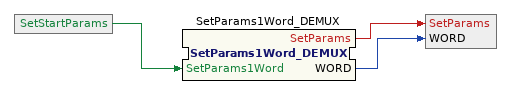
      [picture p97: application VDMA_Station1_CodeGenDistributed.RobotSetStartParams]
      FBS
        SetParams1Word_DEMUX : SetParams1Word_DEMUX;
      END_FBS
      EVENT_CONNECTIONS
        SetParams1Word_DEMUX.SetParams TO SetParams;
      END_CONNECTIONS
      DATA_CONNECTIONS
        SetParams1Word_DEMUX.WORD TO WORD;
      END_CONNECTIONS
      ADAPTER_CONNECTIONS
        SetStartParams TO SetParams1Word_DEMUX.SetParams1Word;
      END_CONNECTIONS
    END_SUBAPPLICATION
    SUBAPPLICATION TurntableSkill
      EVENT_INPUT
        INIT;
        Table_SetStartParam_REQ;
      END_EVENT
      EVENT_OUTPUT
        INITO;
      END_EVENT
      VAR_INPUT
        Table_SetStartParam_IN : WORD;
      END_VAR
      SOCKETS
        AIAS_Skill : IAS_Skill;
      END_SOCKETS
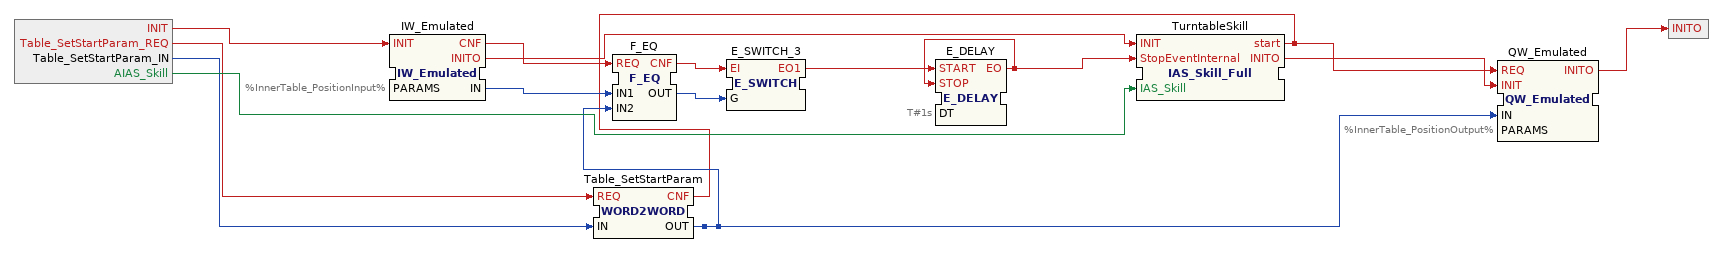
      FBS
        F_EQ : F_EQ;
        E_SWITCH_3 : E_SWITCH;
        Table_SetStartParam : WORD2WORD;
        QW_Emulated : QW_Emulated(PARAMS := %InnerTable_PositionOutput%);
        TurntableSkill : IAS_Skill_Full;
        IW_Emulated : IW_Emulated(PARAMS := %InnerTable_PositionInput%);
        E_DELAY : E_DELAY(DT := T#1s);
      END_FBS
      EVENT_CONNECTIONS
        IW_Emulated.CNF TO F_EQ.REQ;
        TurntableSkill.start TO F_EQ.REQ;
        Table_SetStartParam.CNF TO F_EQ.REQ;
        F_EQ.CNF TO E_SWITCH_3.EI;
        TurntableSkill.start TO QW_Emulated.REQ;
        Table_SetStartParam_REQ TO Table_SetStartParam.REQ;
        INIT TO IW_Emulated.INIT;
        IW_Emulated.INITO TO TurntableSkill.INIT;
        TurntableSkill.INITO TO QW_Emulated.INIT;
        QW_Emulated.INITO TO INITO;
        E_SWITCH_3.EO1 TO E_DELAY.START;
        E_DELAY.EO TO TurntableSkill.StopEventInternal;
        E_DELAY.EO TO E_DELAY.STOP;
      END_CONNECTIONS
      DATA_CONNECTIONS
        IW_Emulated.IN TO F_EQ.IN1;
        Table_SetStartParam.OUT TO F_EQ.IN2;
        F_EQ.OUT TO E_SWITCH_3.G;
        Table_SetStartParam.OUT TO QW_Emulated.IN;
        Table_SetStartParam_IN TO Table_SetStartParam.IN;
      END_CONNECTIONS
      ADAPTER_CONNECTIONS
        AIAS_Skill TO TurntableSkill.IAS_Skill;
      END_CONNECTIONS
    END_SUBAPPLICATION
    SUBAPPLICATION GripperSkill
      EVENT_INPUT
        INIT;
      END_EVENT
      EVENT_OUTPUT
        INITO;
      END_EVENT
      SOCKETS
        AIAS_Skill : IAS_Skill;
      END_SOCKETS
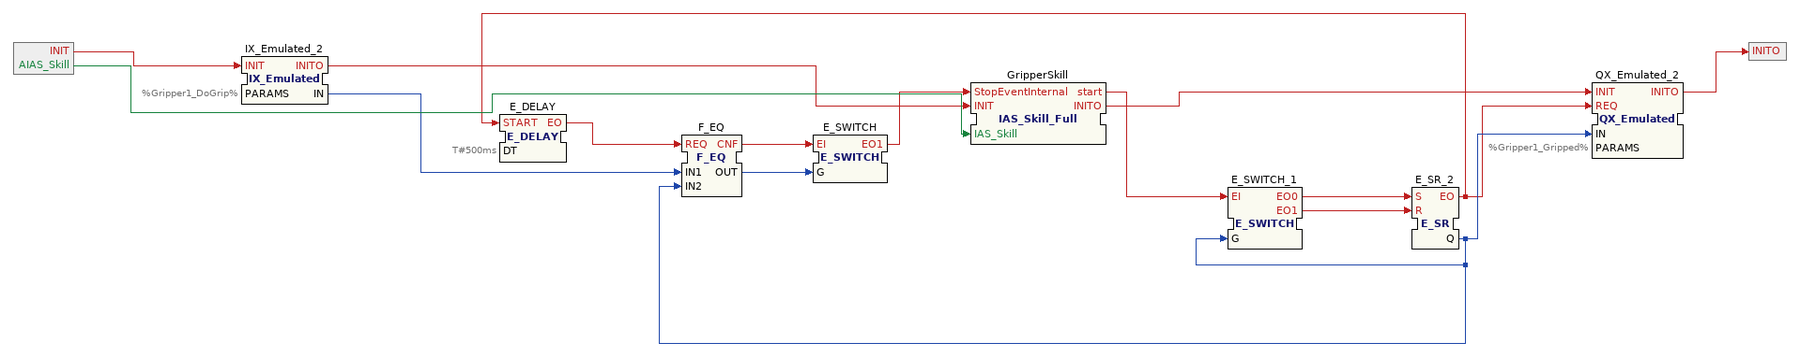
      FBS
        GripperSkill : IAS_Skill_Full;
        F_EQ : F_EQ;
        E_SWITCH_1 : E_SWITCH;
        IX_Emulated_2 : IX_Emulated(PARAMS := %Gripper1_DoGrip%);
        E_DELAY : E_DELAY(DT := T#500ms);
        E_SWITCH : E_SWITCH;
        E_SR_2 : E_SR;
        QX_Emulated_2 : QX_Emulated(PARAMS := %Gripper1_Gripped%);
      END_FBS
      EVENT_CONNECTIONS
        E_SWITCH.EO1 TO GripperSkill.StopEventInternal;
        GripperSkill.start TO E_SWITCH_1.EI;
        E_DELAY.EO TO F_EQ.REQ;
        F_EQ.CNF TO E_SWITCH.EI;
        E_SWITCH_1.EO0 TO E_SR_2.S;
        E_SWITCH_1.EO1 TO E_SR_2.R;
        E_SR_2.EO TO E_DELAY.START;
        INIT TO IX_Emulated_2.INIT;
        IX_Emulated_2.INITO TO GripperSkill.INIT;
        GripperSkill.INITO TO QX_Emulated_2.INIT;
        QX_Emulated_2.INITO TO INITO;
        E_SR_2.EO TO QX_Emulated_2.REQ;
      END_CONNECTIONS
      DATA_CONNECTIONS
        IX_Emulated_2.IN TO F_EQ.IN1;
        E_SR_2.Q TO F_EQ.IN2;
        F_EQ.OUT TO E_SWITCH.G;
        E_SR_2.Q TO E_SWITCH_1.G;
        E_SR_2.Q TO QX_Emulated_2.IN;
      END_CONNECTIONS
      ADAPTER_CONNECTIONS
        AIAS_Skill TO GripperSkill.IAS_Skill;
      END_CONNECTIONS
    END_SUBAPPLICATION
    SUBAPPLICATION RobotSkill
      EVENT_INPUT
        INIT;
        SetStartParam_REQ;
      END_EVENT
      EVENT_OUTPUT
        INITO;
      END_EVENT
      VAR_INPUT
        Robot_SetStartParam_IN : WORD;
      END_VAR
      SOCKETS
        AIAS_Skill : IAS_Skill;
      END_SOCKETS
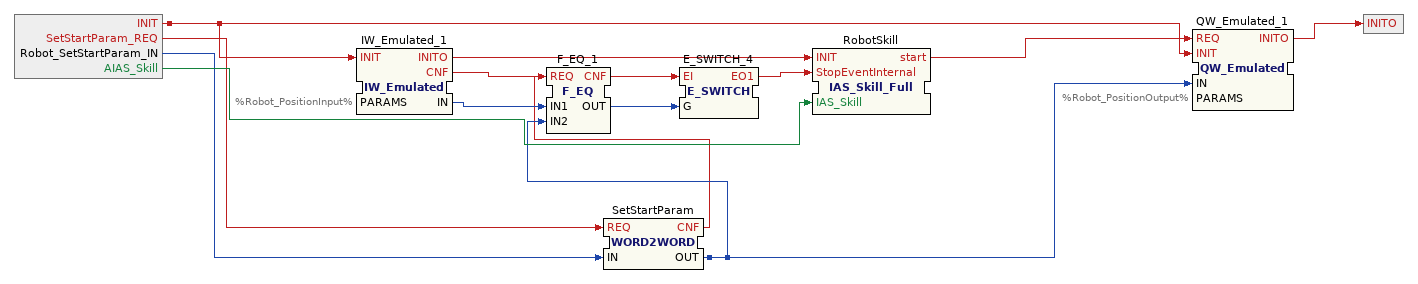
      FBS
        RobotSkill : IAS_Skill_Full;
        IW_Emulated_1 : IW_Emulated(PARAMS := %Robot_PositionInput%);
        E_SWITCH_4 : E_SWITCH;
        F_EQ_1 : F_EQ;
        QW_Emulated_1 : QW_Emulated(PARAMS := %Robot_PositionOutput%);
        SetStartParam : WORD2WORD;
      END_FBS
      EVENT_CONNECTIONS
        IW_Emulated_1.INITO TO RobotSkill.INIT;
        E_SWITCH_4.EO1 TO RobotSkill.StopEventInternal;
        RobotSkill.start TO QW_Emulated_1.REQ;
        IW_Emulated_1.CNF TO F_EQ_1.REQ;
        F_EQ_1.CNF TO E_SWITCH_4.EI;
        SetStartParam.CNF TO F_EQ_1.REQ;
        INIT TO IW_Emulated_1.INIT;
        SetStartParam_REQ TO SetStartParam.REQ;
        QW_Emulated_1.INITO TO INITO;
        INIT TO QW_Emulated_1.INIT;
      END_CONNECTIONS
      DATA_CONNECTIONS
        IW_Emulated_1.IN TO F_EQ_1.IN1;
        F_EQ_1.OUT TO E_SWITCH_4.G;
        SetStartParam.OUT TO F_EQ_1.IN2;
        SetStartParam.OUT TO QW_Emulated_1.IN;
        Robot_SetStartParam_IN TO SetStartParam.IN;
      END_CONNECTIONS
      ADAPTER_CONNECTIONS
        AIAS_Skill TO RobotSkill.IAS_Skill;
      END_CONNECTIONS
    END_SUBAPPLICATION
    SUBAPPLICATION StorageSkill
      EVENT_INPUT
        INIT;
      END_EVENT
      EVENT_OUTPUT
        INITO;
      END_EVENT
      SOCKETS
        AIAS_Skill : IAS_Skill;
      END_SOCKETS
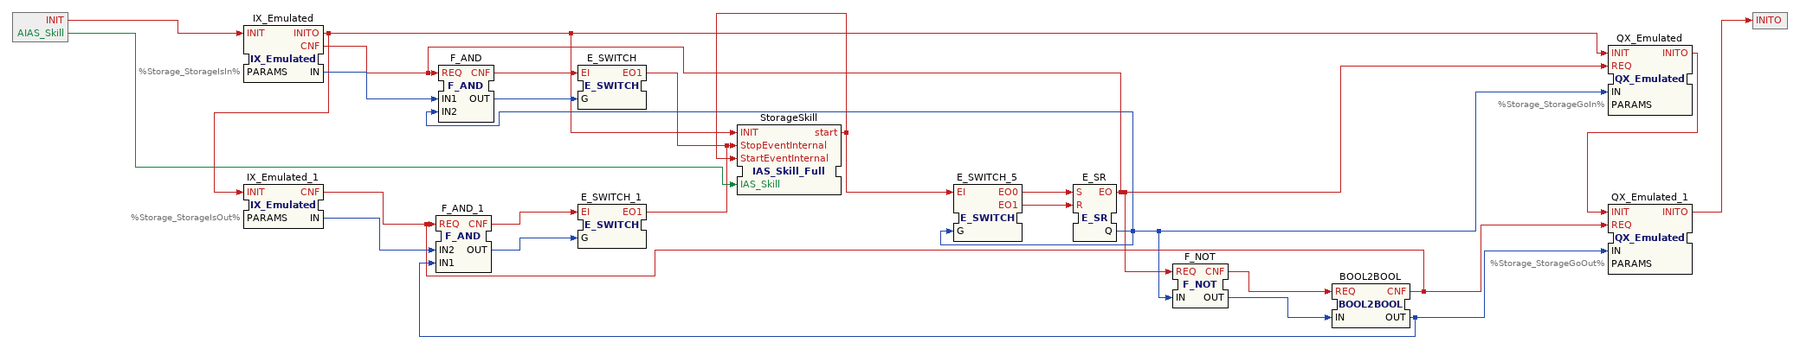
      FBS
        E_SWITCH_5 : E_SWITCH;
        IX_Emulated : IX_Emulated(PARAMS := %Storage_StorageIsIn%);
        F_NOT : F_NOT;
        IX_Emulated_1 : IX_Emulated(PARAMS := %Storage_StorageIsOut%);
        E_SWITCH : E_SWITCH;
        E_SWITCH_1 : E_SWITCH;
        StorageSkill : IAS_Skill_Full;
        F_AND : F_AND;
        BOOL2BOOL : BOOL2BOOL;
        F_AND_1 : F_AND;
        E_SR : E_SR;
        QX_Emulated_1 : QX_Emulated(PARAMS := %Storage_StorageGoOut%);
        QX_Emulated : QX_Emulated(PARAMS := %Storage_StorageGoIn%);
      END_FBS
      EVENT_CONNECTIONS
        StorageSkill.start TO E_SWITCH_5.EI;
        E_SWITCH_5.EO0 TO E_SR.S;
        E_SWITCH_5.EO1 TO E_SR.R;
        IX_Emulated.INITO TO IX_Emulated_1.INIT;
        IX_Emulated.INITO TO StorageSkill.INIT;
        IX_Emulated.CNF TO F_AND.REQ;
        E_SR.EO TO F_NOT.REQ;
        F_NOT.CNF TO BOOL2BOOL.REQ;
        IX_Emulated_1.CNF TO F_AND_1.REQ;
        F_AND.CNF TO E_SWITCH.EI;
        E_SWITCH.EO1 TO StorageSkill.StopEventInternal;
        F_AND_1.CNF TO E_SWITCH_1.EI;
        E_SWITCH_1.EO1 TO StorageSkill.StopEventInternal;
        StorageSkill.start TO StorageSkill.StartEventInternal;
        E_SR.EO TO F_AND.REQ;
        BOOL2BOOL.CNF TO F_AND_1.REQ;
        INIT TO IX_Emulated.INIT;
        QX_Emulated_1.INITO TO INITO;
        IX_Emulated.INITO TO QX_Emulated.INIT;
        QX_Emulated.INITO TO QX_Emulated_1.INIT;
        BOOL2BOOL.CNF TO QX_Emulated_1.REQ;
        E_SR.EO TO QX_Emulated.REQ;
      END_CONNECTIONS
      DATA_CONNECTIONS
        E_SR.Q TO E_SWITCH_5.G;
        IX_Emulated.IN TO F_AND.IN1;
        E_SR.Q TO F_NOT.IN;
        F_NOT.OUT TO BOOL2BOOL.IN;
        IX_Emulated_1.IN TO F_AND_1.IN2;
        F_AND.OUT TO E_SWITCH.G;
        F_AND_1.OUT TO E_SWITCH_1.G;
        E_SR.Q TO F_AND.IN2;
        BOOL2BOOL.OUT TO F_AND_1.IN1;
        E_SR.Q TO QX_Emulated.IN;
        BOOL2BOOL.OUT TO QX_Emulated_1.IN;
      END_CONNECTIONS
      ADAPTER_CONNECTIONS
        AIAS_Skill TO StorageSkill.IAS_Skill;
      END_CONNECTIONS
    END_SUBAPPLICATION
    EVENT_CONNECTIONS
      StorageSkill.INITO TO TurntableSkill.INIT;
      TurntableSkill.INITO TO GripperSkill.INIT;
      RobotSetStartParams.SetParams TO RobotSkill.SetStartParam_REQ;
      GripperSkill.INITO TO RobotSkill.INIT;
      TurnTableSetStartParams.SetParams TO TurntableSkill.Table_SetStartParam_REQ;
      Orchestrator.doRndCnt TO Orchestrator.rndCntDone;
      Orchestrator.doRepCnt TO Orchestrator.repCntDone;
    END_CONNECTIONS
    DATA_CONNECTIONS
      TurnTableSetStartParams.WORD TO TurntableSkill.Table_SetStartParam_IN;
      RobotSetStartParams.WORD TO RobotSkill.Robot_SetStartParam_IN;
    END_CONNECTIONS
    ADAPTER_CONNECTIONS
      Orchestrator.StorageSkill_IAS_Skill TO StorageSkill.AIAS_Skill;
      Orchestrator.TurnTableSetStartParams_SetParams1Word TO TurnTableSetStartParams.SetStartParams;
      Orchestrator.TurntableSkill_IAS_Skill TO TurntableSkill.AIAS_Skill;
      Orchestrator.RobotSetStartParams_SetParams1Word TO RobotSetStartParams.SetStartParams;
      Orchestrator.RobotSkill_IAS_Skill TO RobotSkill.AIAS_Skill;
      Orchestrator.GripperSkill_IAS_Skill TO GripperSkill.AIAS_Skill;
    END_CONNECTIONS
  END_APPLICATION
  APPLICATION VDMA_Station1_DA
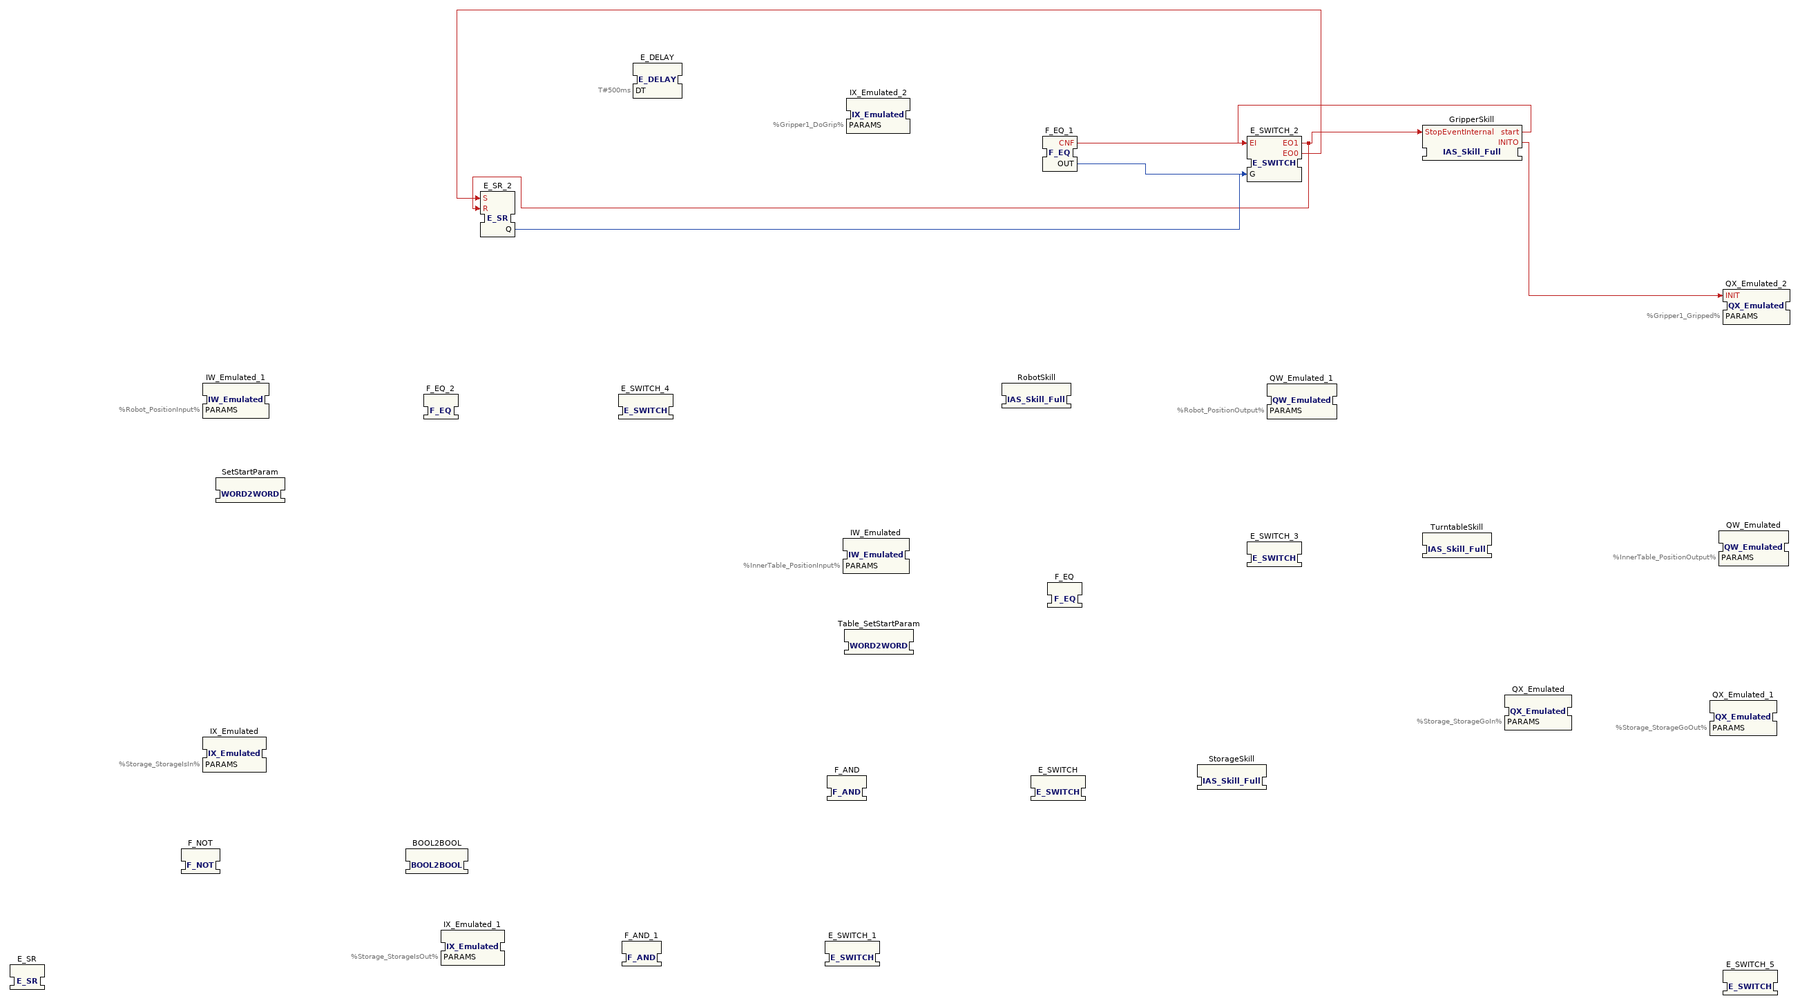
    FBS
      E_SWITCH_5 : E_SWITCH;
      IX_Emulated : IX_Emulated(PARAMS := %Storage_StorageIsIn%);
      F_NOT : F_NOT;
      IX_Emulated_1 : IX_Emulated(PARAMS := %Storage_StorageIsOut%);
      E_SWITCH : E_SWITCH;
      E_SWITCH_1 : E_SWITCH;
      StorageSkill : IAS_Skill_Full;
      F_AND : F_AND;
      BOOL2BOOL : BOOL2BOOL;
      F_AND_1 : F_AND;
      E_SR : E_SR;
      F_EQ : F_EQ;
      E_SWITCH_3 : E_SWITCH;
      Table_SetStartParam : WORD2WORD;
      QW_Emulated : QW_Emulated(PARAMS := %InnerTable_PositionOutput%);
      TurntableSkill : IAS_Skill_Full;
      IW_Emulated : IW_Emulated(PARAMS := %InnerTable_PositionInput%);
      GripperSkill : IAS_Skill_Full;
      F_EQ_1 : F_EQ;
      E_SWITCH_2 : E_SWITCH;
      IX_Emulated_2 : IX_Emulated(PARAMS := %Gripper1_DoGrip%);
      E_DELAY : E_DELAY(DT := T#500ms);
      E_SWITCH_2 : E_SWITCH;
      E_SR_2 : E_SR;
      RobotSkill : IAS_Skill_Full;
      IW_Emulated_1 : IW_Emulated(PARAMS := %Robot_PositionInput%);
      E_SWITCH_4 : E_SWITCH;
      F_EQ_2 : F_EQ;
      QW_Emulated_1 : QW_Emulated(PARAMS := %Robot_PositionOutput%);
      SetStartParam : WORD2WORD;
      QX_Emulated_2 : QX_Emulated(PARAMS := %Gripper1_Gripped%);
      QX_Emulated_1 : QX_Emulated(PARAMS := %Storage_StorageGoOut%);
      QX_Emulated : QX_Emulated(PARAMS := %Storage_StorageGoIn%);
    END_FBS
    EVENT_CONNECTIONS
      E_SWITCH_2.EO1 TO GripperSkill.StopEventInternal;
      GripperSkill.start TO E_SWITCH_2.EI;
      F_EQ_1.CNF TO E_SWITCH_2.EI;
      E_SWITCH_2.EO0 TO E_SR_2.S;
      E_SWITCH_2.EO1 TO E_SR_2.R;
      GripperSkill.INITO TO QX_Emulated_2.INIT;
    END_CONNECTIONS
    DATA_CONNECTIONS
      F_EQ_1.OUT TO E_SWITCH_2.G;
      E_SR_2.Q TO E_SWITCH_2.G;
    END_CONNECTIONS
  END_APPLICATION
  DEVICE Robot : FORTE_PC(MGR_ID := "localhost:61499")
    {SET_ATTRIBUTE(Profile, HOLOBLOC)} (* device profile *)
    RESOURCE central : EMB_RES
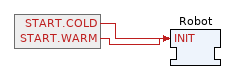
      SUBAPPLICATION Robot
        EVENT_INPUT
          INIT;
        END_EVENT
      END_SUBAPPLICATION
      EVENT_CONNECTIONS
        START.COLD TO Robot.INIT;
        START.WARM TO Robot.INIT;
      END_CONNECTIONS
    END_RESOURCE
    RESOURCE decentral : EMB_RES
    END_RESOURCE
  END_DEVICE
  DEVICE InnerTable : FORTE_PC(MGR_ID := "localhost:61500")
    {SET_ATTRIBUTE(Profile, HOLOBLOC)} (* device profile *)
    RESOURCE central : EMB_RES
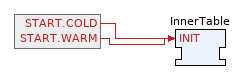
      SUBAPPLICATION InnerTable
        EVENT_INPUT
          INIT;
        END_EVENT
      END_SUBAPPLICATION
      EVENT_CONNECTIONS
        START.COLD TO InnerTable.INIT;
        START.WARM TO InnerTable.INIT;
      END_CONNECTIONS
    END_RESOURCE
    RESOURCE decentral : EMB_RES
    END_RESOURCE
  END_DEVICE
  DEVICE Storage : FORTE_PC(MGR_ID := "localhost:61501")
    {SET_ATTRIBUTE(Profile, HOLOBLOC)} (* device profile *)
    RESOURCE central : EMB_RES
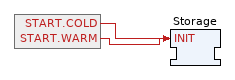
      SUBAPPLICATION Storage
        EVENT_INPUT
          INIT;
        END_EVENT
      END_SUBAPPLICATION
      EVENT_CONNECTIONS
        START.COLD TO Storage.INIT;
        START.WARM TO Storage.INIT;
      END_CONNECTIONS
    END_RESOURCE
    RESOURCE decentral : EMB_RES
    END_RESOURCE
  END_DEVICE
  DEVICE Gripper1 : FORTE_PC(MGR_ID := "localhost:61502")
    {SET_ATTRIBUTE(Profile, HOLOBLOC)} (* device profile *)
    RESOURCE central : EMB_RES
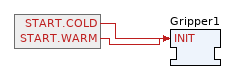
      SUBAPPLICATION Gripper1
        EVENT_INPUT
          INIT;
        END_EVENT
      END_SUBAPPLICATION
      EVENT_CONNECTIONS
        START.COLD TO Gripper1.INIT;
        START.WARM TO Gripper1.INIT;
      END_CONNECTIONS
    END_RESOURCE
    RESOURCE decentral : EMB_RES
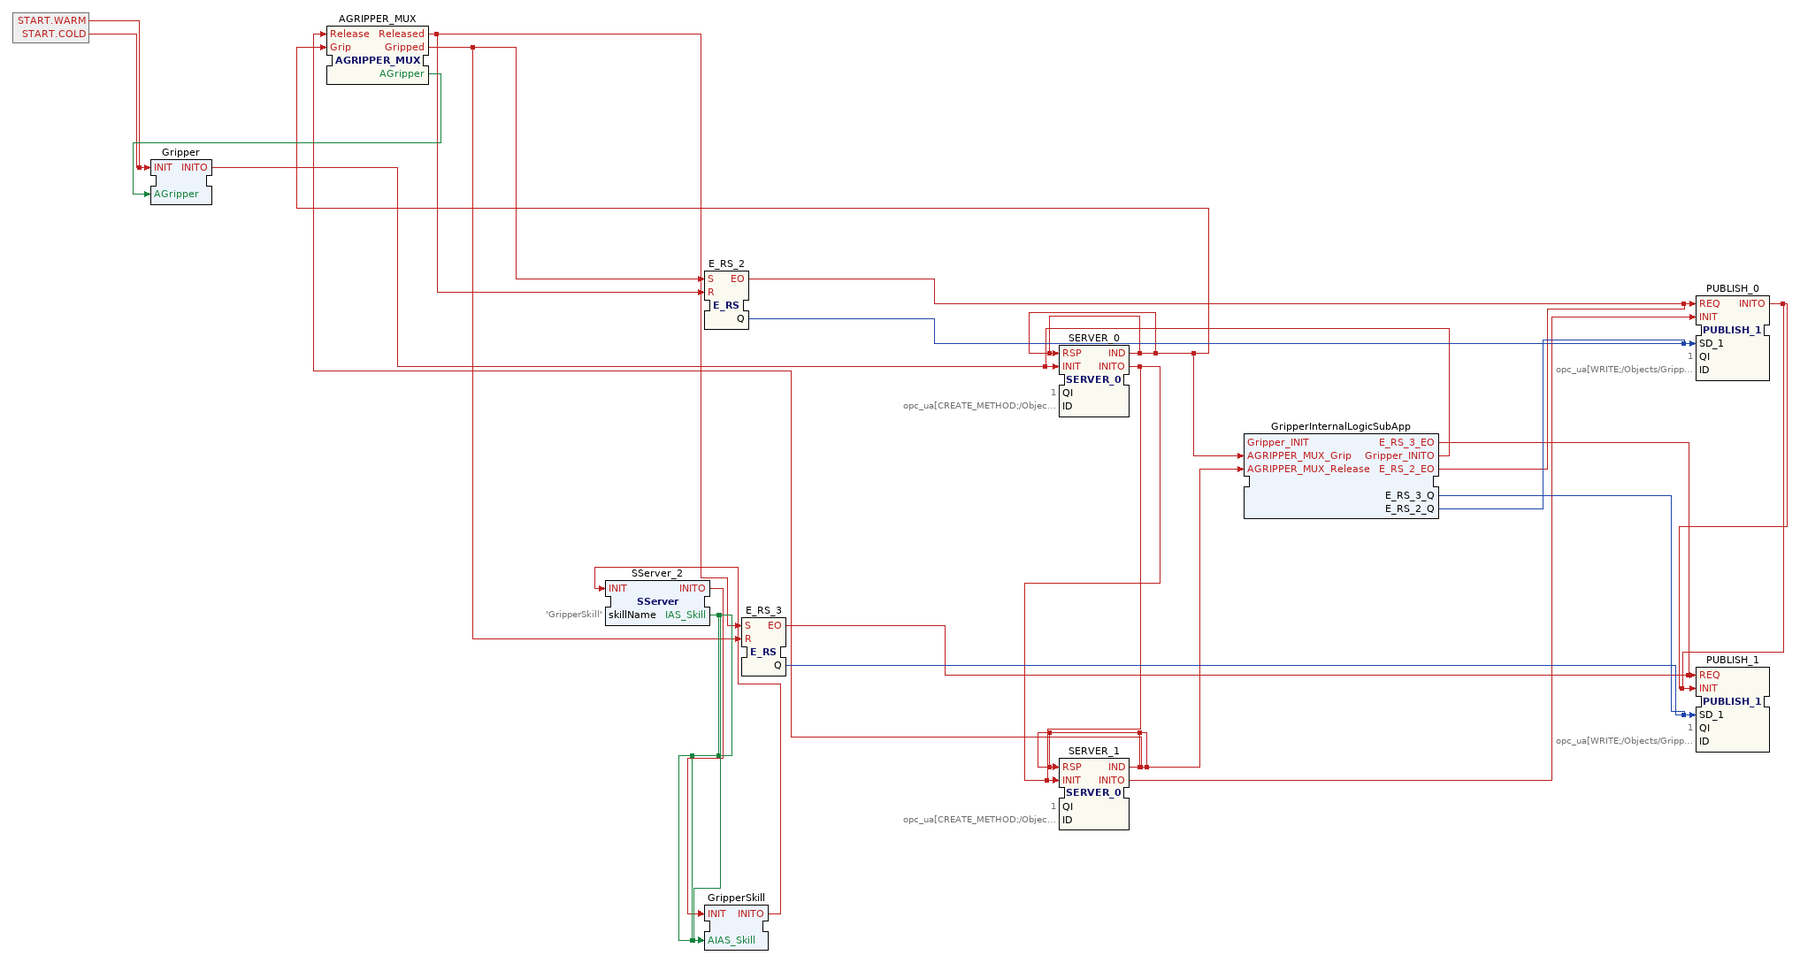
      FBS
        SERVER_1 : SERVER_0(QI := 1, ID := opc_ua[CREATE_METHOD;/Objects/Gripper/Release]);
        PUBLISH_1 : PUBLISH_1(QI := 1, ID := opc_ua[WRITE;/Objects/Gripper/Released]);
        AGRIPPER_MUX : AGRIPPER_MUX;
        E_RS_3 : E_RS;
        SERVER_0 : SERVER_0(QI := 1, ID := opc_ua[CREATE_METHOD;/Objects/Gripper/Grip]);
        E_RS_2 : E_RS;
        PUBLISH_0 : PUBLISH_1(QI := 1, ID := opc_ua[WRITE;/Objects/Gripper/Gripped]);
        SERVER_1 : SERVER_0(QI := 1, ID := opc_ua[CREATE_METHOD;/Objects/Gripper/Release]);
        PUBLISH_0 : PUBLISH_1(QI := 1, ID := opc_ua[WRITE;/Objects/Gripper/Gripped]);
        SERVER_0 : SERVER_0(QI := 1, ID := opc_ua[CREATE_METHOD;/Objects/Gripper/Grip]);
        PUBLISH_1 : PUBLISH_1(QI := 1, ID := opc_ua[WRITE;/Objects/Gripper/Released]);
      END_FBS
      SUBAPPS
        SServer_2 : SServer;
        SServer_2 : SServer_;
        SServer_2 : SServer(skillName := 'GripperSkill');
      END_SUBAPPS
      SUBAPPLICATION GripperSkill
        EVENT_INPUT
          INIT;
        END_EVENT
        EVENT_OUTPUT
          INITO;
        END_EVENT
        SOCKETS
          AIAS_Skill : IAS_Skill;
        END_SOCKETS
      END_SUBAPPLICATION
      SUBAPPLICATION Gripper
        EVENT_INPUT
          INIT;
        END_EVENT
        EVENT_OUTPUT
          INITO;
        END_EVENT
        SOCKETS
          AGripper : AGripper;
        END_SOCKETS
      END_SUBAPPLICATION
      SUBAPPLICATION GripperInternalLogicSubApp
        EVENT_INPUT
          Gripper_INIT;
          AGRIPPER_MUX_Grip;
          AGRIPPER_MUX_Release;
        END_EVENT
        EVENT_OUTPUT
          E_RS_3_EO;
          Gripper_INITO;
          E_RS_2_EO;
        END_EVENT
        VAR_OUTPUT
          E_RS_3_Q : BOOL;
          E_RS_2_Q : BOOL;
        END_VAR
      END_SUBAPPLICATION
      EVENT_CONNECTIONS
        GripperSkill.INITO TO SServer_2.INIT;
        SERVER_1.IND TO SERVER_1.RSP;
        SERVER_1.IND TO AGRIPPER_MUX.Release;
        E_RS_3.EO TO PUBLISH_1.REQ;
        AGRIPPER_MUX.Released TO E_RS_3.S;
        AGRIPPER_MUX.Gripped TO E_RS_3.R;
        START.WARM TO Gripper.INIT;
        START.COLD TO Gripper.INIT;
        SERVER_0.IND TO SERVER_0.RSP;
        SERVER_0.IND TO AGRIPPER_MUX.Grip;
        SERVER_0.INITO TO SERVER_1.INIT;
        Gripper.INITO TO SERVER_0.INIT;
        AGRIPPER_MUX.Gripped TO E_RS_2.S;
        AGRIPPER_MUX.Released TO E_RS_2.R;
        PUBLISH_0.INITO TO PUBLISH_1.INIT;
        E_RS_2.EO TO PUBLISH_0.REQ;
        SERVER_1.INITO TO PUBLISH_0.INIT;
        GripperSkill.INITO TO SServer_2.INIT;
        SServer_2.INITO TO GripperSkill.INIT;
        SERVER_1.IND TO SERVER_1.RSP;
        SERVER_1.INITO TO PUBLISH_0.INIT;
        SERVER_0.IND TO SERVER_0.RSP;
        SERVER_0.INITO TO SERVER_1.INIT;
        PUBLISH_0.INITO TO PUBLISH_1.INIT;
        SERVER_0.IND TO GripperInternalLogicSubApp.AGRIPPER_MUX_Grip;
        SERVER_1.IND TO GripperInternalLogicSubApp.AGRIPPER_MUX_Release;
        GripperInternalLogicSubApp.E_RS_3_EO TO PUBLISH_1.REQ;
        GripperInternalLogicSubApp.Gripper_INITO TO SERVER_0.INIT;
        GripperInternalLogicSubApp.E_RS_2_EO TO PUBLISH_0.REQ;
        GripperSkill.INITO TO SServer_2.INIT;
        SServer_2.INITO TO GripperSkill.INIT;
      END_CONNECTIONS
      DATA_CONNECTIONS
        E_RS_3.Q TO PUBLISH_1.SD_1;
        E_RS_2.Q TO PUBLISH_0.SD_1;
        GripperInternalLogicSubApp.E_RS_3_Q TO PUBLISH_1.SD_1;
        GripperInternalLogicSubApp.E_RS_2_Q TO PUBLISH_0.SD_1;
      END_CONNECTIONS
      ADAPTER_CONNECTIONS
        SServer_2.IAS_Skill TO GripperSkill.AIAS_Skill;
        SServer_2.IAS_Skill TO GripperSkill.AIAS_Skill;
        AGRIPPER_MUX.AGripper TO Gripper.AGripper;
        SServer_2.IAS_Skill TO GripperSkill.AIAS_Skill;
        SServer_2.IAS_Skill TO GripperSkill.AIAS_Skill;
      END_CONNECTIONS
    END_RESOURCE
  END_DEVICE
  DEVICE Gripper2 : FORTE_PC(MGR_ID := "localhost:61503")
    {SET_ATTRIBUTE(Profile, HOLOBLOC)} (* device profile *)
    RESOURCE EMB_RES : EMB_RES
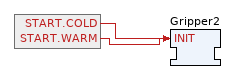
      SUBAPPLICATION Gripper2
        EVENT_INPUT
          INIT;
        END_EVENT
      END_SUBAPPLICATION
      EVENT_CONNECTIONS
        START.COLD TO Gripper2.INIT;
        START.WARM TO Gripper2.INIT;
      END_CONNECTIONS
    END_RESOURCE
  END_DEVICE
  DEVICE IOs_to_OPCUA : FORTE_PC(MGR_ID := "localhost:61515")
    {SET_ATTRIBUTE(Profile, HOLOBLOC)} (* device profile *)
    RESOURCE EMB_RES : EMB_RES
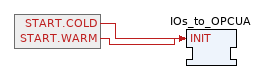
      SUBAPPLICATION IOs_to_OPCUA
        EVENT_INPUT
          INIT;
        END_EVENT
      END_SUBAPPLICATION
      EVENT_CONNECTIONS
        START.COLD TO IOs_to_OPCUA.INIT;
        START.WARM TO IOs_to_OPCUA.INIT;
      END_CONNECTIONS
    END_RESOURCE
  END_DEVICE
  DEVICE hierControl : FORTE_PC(MGR_ID := "localhost:61504")
    {SET_ATTRIBUTE(Profile, HOLOBLOC)} (* device profile *)
    RESOURCE central : EMB_RES
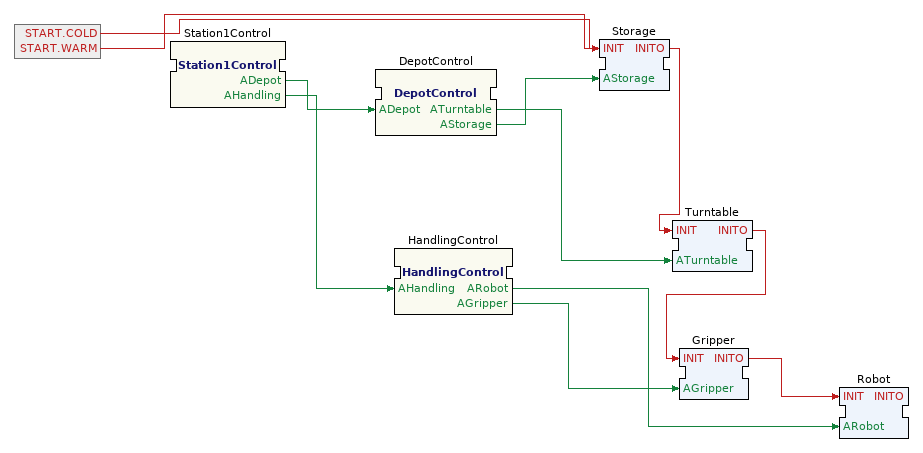
      FBS
        HandlingControl : HandlingControl;
        DepotControl : DepotControl;
        Station1Control : Station1Control;
      END_FBS
      SUBAPPLICATION Robot
        EVENT_INPUT
          INIT;
        END_EVENT
        EVENT_OUTPUT
          INITO;
        END_EVENT
        SOCKETS
          ARobot : ARobot;
        END_SOCKETS
      END_SUBAPPLICATION
      SUBAPPLICATION Gripper
        EVENT_INPUT
          INIT;
        END_EVENT
        EVENT_OUTPUT
          INITO;
        END_EVENT
        SOCKETS
          AGripper : AGripper;
        END_SOCKETS
      END_SUBAPPLICATION
      SUBAPPLICATION Turntable
        EVENT_INPUT
          INIT;
        END_EVENT
        EVENT_OUTPUT
          INITO;
        END_EVENT
        SOCKETS
          ATurntable : ATurntable;
        END_SOCKETS
      END_SUBAPPLICATION
      SUBAPPLICATION Storage
        EVENT_INPUT
          INIT;
        END_EVENT
        EVENT_OUTPUT
          INITO;
        END_EVENT
        SOCKETS
          AStorage : AStorage;
        END_SOCKETS
      END_SUBAPPLICATION
      EVENT_CONNECTIONS
        Gripper.INITO TO Robot.INIT;
        Turntable.INITO TO Gripper.INIT;
        Storage.INITO TO Turntable.INIT;
        START.COLD TO Storage.INIT;
        START.WARM TO Storage.INIT;
      END_CONNECTIONS
      ADAPTER_CONNECTIONS
        HandlingControl.ARobot TO Robot.ARobot;
        HandlingControl.AGripper TO Gripper.AGripper;
        DepotControl.ATurntable TO Turntable.ATurntable;
        DepotControl.AStorage TO Storage.AStorage;
        Station1Control.ADepot TO DepotControl.ADepot;
        Station1Control.AHandling TO HandlingControl.AHandling;
      END_CONNECTIONS
    END_RESOURCE
    RESOURCE decentral : EMB_RES
      FBS
        DepotControl : DepotControl;
        Station1Control : Station1Control;
        HandlingControl : HandlingControl;
        CLIENT_0 : CLIENT_0(QI := 1, ID := opc_ua[CALL_METHOD;opc.tcp://localhost:4842#;/Objects/Storage/GoIn]);
        CLIENT_5 : CLIENT_0(QI := 1, ID := opc_ua[CALL_METHOD;opc.tcp://localhost:4843#;/Objects/Gripper/Release]);
        CLIENT_4 : CLIENT_0(QI := 1, ID := opc_ua[CALL_METHOD;opc.tcp://localhost:4843#;/Objects/Gripper/Grip]);
        RobotSubApp : AROBOT_DEMUX;
        SUBSCRIBE_1 : SUBSCRIBE_1(QI := 1, ID := opc_ua[SUBSCRIBE;opc.tcp://localhost:4840#;/Objects/Robot/CurrentPosition]);
        SUBSCRIBE_2 : SUBSCRIBE_1(QI := 1, ID := opc_ua[SUBSCRIBE;opc.tcp://localhost:4841#;/Objects/Turntable/CurrentPosition]);
        TurntableSubApp : ATURNTABLE_DEMUX;
        SUBSCRIBE_3 : SUBSCRIBE_1(QI := 1, ID := opc_ua[SUBSCRIBE;opc.tcp://localhost:4842#;/Objects/Storage/IsOut]);
        SUBSCRIBE_9 : SUBSCRIBE_1(QI := 1, ID := opc_ua[SUBSCRIBE;opc.tcp://localhost:4842#;/Objects/Storage/IsIn]);
        E_SWITCH_1 : E_SWITCH;
        E_SWITCH : E_SWITCH;
        SUBSCRIBE_4 : SUBSCRIBE_1(QI := 1, ID := opc_ua[SUBSCRIBE;opc.tcp://localhost:4843#;/Objects/Gripper/Gripped]);
        SUBSCRIBE_5 : SUBSCRIBE_1(QI := 1, ID := opc_ua[SUBSCRIBE;opc.tcp://localhost:4843#;/Objects/Gripper/Released]);
        E_SWITCH_2 : E_SWITCH;
        E_SWITCH_3 : E_SWITCH;
        CLIENT_2 : CLIENT_1_0(QI := 1, ID := opc_ua[CALL_METHOD;opc.tcp://localhost:4841#;/Objects/Turntable/NewPosition]);
        CLIENT_1 : CLIENT_1_0(QI := 1, ID := opc_ua[CALL_METHOD;opc.tcp://localhost:4840#;/Objects/Robot/PresetPositionUpd]);
        CLIENT_3 : CLIENT_0(QI := 1, ID := opc_ua[CALL_METHOD;opc.tcp://localhost:4842#;/Objects/Storage/GoOut]);
        SUBSCRIBE_5 : SUBSCRIBE_1(QI := 1, ID := opc_ua[SUBSCRIBE;opc.tcp://localhost:4843#;/Objects/Gripper/Released]);
        CLIENT_3 : CLIENT_0(QI := 1, ID := opc_ua[CALL_METHOD;opc.tcp://localhost:4842#;/Objects/Storage/GoOut]);
        SUBSCRIBE_9 : SUBSCRIBE_1(QI := 1, ID := opc_ua[SUBSCRIBE;opc.tcp://localhost:4842#;/Objects/Storage/IsIn]);
        SUBSCRIBE_4 : SUBSCRIBE_1(QI := 1, ID := opc_ua[SUBSCRIBE;opc.tcp://localhost:4843#;/Objects/Gripper/Gripped]);
        SUBSCRIBE_3 : SUBSCRIBE_1(QI := 1, ID := opc_ua[SUBSCRIBE;opc.tcp://localhost:4842#;/Objects/Storage/IsOut]);
        CLIENT_1 : CLIENT_1_0(QI := 1, ID := opc_ua[CALL_METHOD;opc.tcp://localhost:4840#;/Objects/Robot/PresetPositionUpd]);
        CLIENT_2 : CLIENT_1_0(QI := 1, ID := opc_ua[CALL_METHOD;opc.tcp://localhost:4841#;/Objects/Turntable/NewPosition]);
      END_FBS
      SUBAPPLICATION StorageSubApp
        EVENT_INPUT
          E_SWITCH_1_EI;
          E_SWITCH_EI;
        END_EVENT
        EVENT_OUTPUT
          ASTORAGE_DEMUX_GoIn;
          ASTORAGE_DEMUX_GoOut;
        END_EVENT
        VAR_INPUT
          E_SWITCH_1_G : BOOL;
          E_SWITCH_G : BOOL;
        END_VAR
        SOCKETS
          ASTORAGE_DEMUX_AStorage : AStorage;
        END_SOCKETS
      END_SUBAPPLICATION
      SUBAPPLICATION GripperSubApp
        EVENT_INPUT
          E_SWITCH_2_EI;
          E_SWITCH_3_EI;
        END_EVENT
        EVENT_OUTPUT
          AGRIPPER_DEMUX_Grip;
          AGRIPPER_DEMUX_Release;
        END_EVENT
        VAR_INPUT
          E_SWITCH_2_G : BOOL;
          E_SWITCH_3_G : BOOL;
        END_VAR
        SOCKETS
          AGRIPPER_DEMUX_AGripper : AGripper;
        END_SOCKETS
      END_SUBAPPLICATION
      EVENT_CONNECTIONS
        CLIENT_4.INITO TO CLIENT_5.INIT;
        SUBSCRIBE_1.IND TO RobotSubApp.PositionUpdate;
        SUBSCRIBE_2.IND TO TurntableSubApp.PositionUpd;
        SUBSCRIBE_3.INITO TO CLIENT_0.INIT;
        SUBSCRIBE_9.IND TO E_SWITCH_1.EI;
        SUBSCRIBE_3.IND TO E_SWITCH.EI;
        START.COLD TO SUBSCRIBE_9.INIT;
        START.WARM TO SUBSCRIBE_9.INIT;
        SUBSCRIBE_2.INITO TO SUBSCRIBE_4.INIT;
        SUBSCRIBE_4.INITO TO SUBSCRIBE_5.INIT;
        SUBSCRIBE_5.INITO TO CLIENT_4.INIT;
        SUBSCRIBE_5.INITO TO SUBSCRIBE_1.INIT;
        SUBSCRIBE_4.IND TO E_SWITCH_2.EI;
        SUBSCRIBE_5.IND TO E_SWITCH_3.EI;
        SUBSCRIBE_9.INITO TO SUBSCRIBE_3.INIT;
        SUBSCRIBE_2.INITO TO CLIENT_2.INIT;
        TurntableSubApp.NewPosition TO CLIENT_2.REQ;
        SUBSCRIBE_1.INITO TO CLIENT_1.INIT;
        RobotSubApp.PresetPositionUpd TO CLIENT_1.REQ;
        CLIENT_3.INITO TO SUBSCRIBE_2.INIT;
        CLIENT_0.INITO TO CLIENT_3.INIT;
        SUBSCRIBE_5.INITO TO CLIENT_4.INIT;
        SUBSCRIBE_5.INITO TO SUBSCRIBE_1.INIT;
        CLIENT_0.INITO TO CLIENT_3.INIT;
        CLIENT_3.INITO TO SUBSCRIBE_2.INIT;
        SUBSCRIBE_2.INITO TO SUBSCRIBE_4.INIT;
        SUBSCRIBE_4.INITO TO SUBSCRIBE_5.INIT;
        SUBSCRIBE_9.INITO TO SUBSCRIBE_3.INIT;
        SUBSCRIBE_3.INITO TO CLIENT_0.INIT;
        SUBSCRIBE_1.INITO TO CLIENT_1.INIT;
        RobotSubApp.PresetPositionUpd TO CLIENT_1.REQ;
        SUBSCRIBE_2.INITO TO CLIENT_2.INIT;
        TurntableSubApp.NewPosition TO CLIENT_2.REQ;
        SUBSCRIBE_9.IND TO StorageSubApp.E_SWITCH_1_EI;
        SUBSCRIBE_3.IND TO StorageSubApp.E_SWITCH_EI;
        StorageSubApp.ASTORAGE_DEMUX_GoIn TO CLIENT_0.REQ;
        StorageSubApp.ASTORAGE_DEMUX_GoOut TO CLIENT_3.REQ;
        SUBSCRIBE_4.IND TO GripperSubApp.E_SWITCH_2_EI;
        SUBSCRIBE_5.IND TO GripperSubApp.E_SWITCH_3_EI;
        GripperSubApp.AGRIPPER_DEMUX_Grip TO CLIENT_4.REQ;
        GripperSubApp.AGRIPPER_DEMUX_Release TO CLIENT_5.REQ;
      END_CONNECTIONS
      DATA_CONNECTIONS
        SUBSCRIBE_1.RD_1 TO RobotSubApp.CurrentPosition;
        SUBSCRIBE_2.RD_1 TO TurntableSubApp.CurrentPosition;
        SUBSCRIBE_9.RD_1 TO E_SWITCH_1.G;
        SUBSCRIBE_3.RD_1 TO E_SWITCH.G;
        SUBSCRIBE_4.RD_1 TO E_SWITCH_2.G;
        SUBSCRIBE_5.RD_1 TO E_SWITCH_3.G;
        TurntableSubApp.Position TO CLIENT_2.SD_1;
        RobotSubApp.PresetPosition TO CLIENT_1.SD_1;
        RobotSubApp.PresetPosition TO CLIENT_1.SD_1;
        TurntableSubApp.Position TO CLIENT_2.SD_1;
        SUBSCRIBE_9.RD_1 TO StorageSubApp.E_SWITCH_1_G;
        SUBSCRIBE_3.RD_1 TO StorageSubApp.E_SWITCH_G;
        SUBSCRIBE_4.RD_1 TO GripperSubApp.E_SWITCH_2_G;
        SUBSCRIBE_5.RD_1 TO GripperSubApp.E_SWITCH_3_G;
      END_CONNECTIONS
      ADAPTER_CONNECTIONS
        Station1Control.ADepot TO DepotControl.ADepot;
        Station1Control.AHandling TO HandlingControl.AHandling;
        HandlingControl.ARobot TO RobotSubApp.ARobot;
        DepotControl.ATurntable TO TurntableSubApp.ATurntable;
        DepotControl.AStorage TO StorageSubApp.ASTORAGE_DEMUX_AStorage;
        HandlingControl.AGripper TO GripperSubApp.AGRIPPER_DEMUX_AGripper;
      END_CONNECTIONS
    END_RESOURCE
  END_DEVICE
  DEVICE skillControl : FORTE_PC(MGR_ID := "localhost:61505")
    {SET_ATTRIBUTE(Profile, HOLOBLOC)} (* device profile *)
    RESOURCE central : EMB_RES
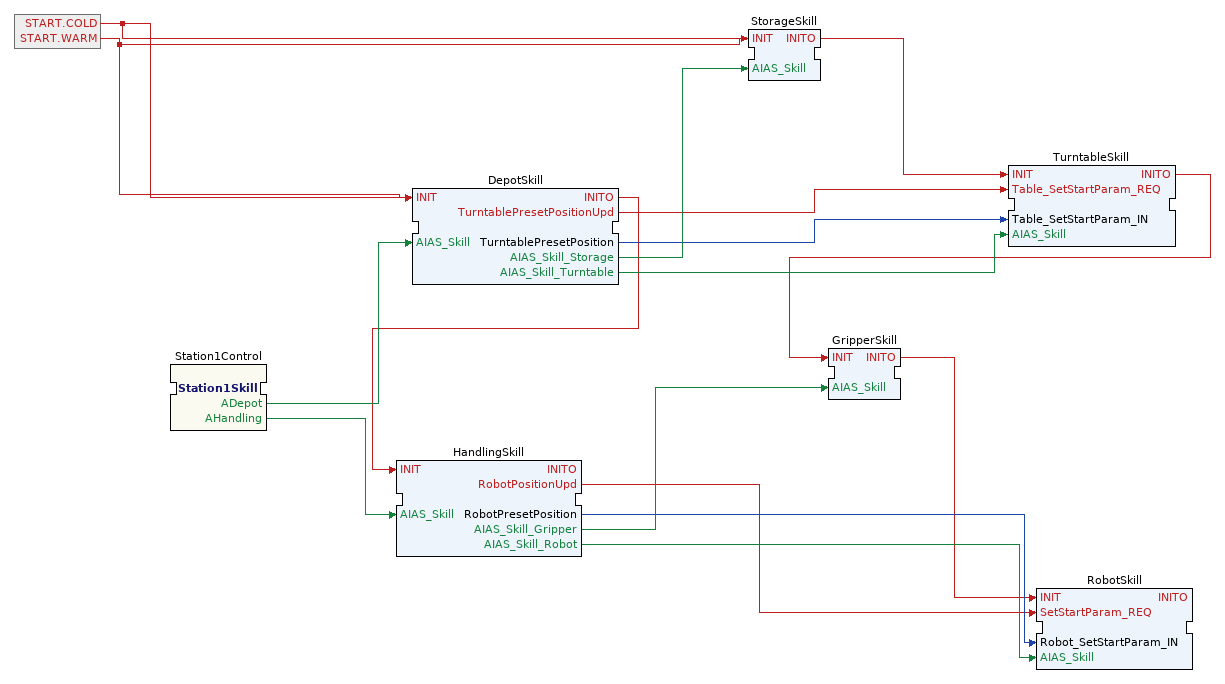
      FBS
        Station1Control : Station1Skill;
      END_FBS
      SUBAPPLICATION StorageSkill
        EVENT_INPUT
          INIT;
        END_EVENT
        EVENT_OUTPUT
          INITO;
        END_EVENT
        SOCKETS
          AIAS_Skill : IAS_Skill;
        END_SOCKETS
      END_SUBAPPLICATION
      SUBAPPLICATION TurntableSkill
        EVENT_INPUT
          INIT;
          Table_SetStartParam_REQ;
        END_EVENT
        EVENT_OUTPUT
          INITO;
        END_EVENT
        VAR_INPUT
          Table_SetStartParam_IN : WORD;
        END_VAR
        SOCKETS
          AIAS_Skill : IAS_Skill;
        END_SOCKETS
      END_SUBAPPLICATION
      SUBAPPLICATION DepotSkill
        EVENT_INPUT
          INIT;
        END_EVENT
        EVENT_OUTPUT
          INITO;
          TurntablePresetPositionUpd;
        END_EVENT
        VAR_OUTPUT
          TurntablePresetPosition : WORD;
        END_VAR
        SOCKETS
          AIAS_Skill : IAS_Skill;
        END_SOCKETS
        PLUGS
          AIAS_Skill_Storage : IAS_Skill;
          AIAS_Skill_Turntable : IAS_Skill;
        END_PLUGS
      END_SUBAPPLICATION
      SUBAPPLICATION GripperSkill
        EVENT_INPUT
          INIT;
        END_EVENT
        EVENT_OUTPUT
          INITO;
        END_EVENT
        SOCKETS
          AIAS_Skill : IAS_Skill;
        END_SOCKETS
      END_SUBAPPLICATION
      SUBAPPLICATION HandlingSkill
        EVENT_INPUT
          INIT;
        END_EVENT
        EVENT_OUTPUT
          INITO;
          RobotPositionUpd;
        END_EVENT
        VAR_OUTPUT
          RobotPresetPosition : WORD;
        END_VAR
        SOCKETS
          AIAS_Skill : IAS_Skill;
        END_SOCKETS
        PLUGS
          AIAS_Skill_Gripper : IAS_Skill;
          AIAS_Skill_Robot : IAS_Skill;
        END_PLUGS
      END_SUBAPPLICATION
      SUBAPPLICATION RobotSkill
        EVENT_INPUT
          INIT;
          SetStartParam_REQ;
        END_EVENT
        EVENT_OUTPUT
          INITO;
        END_EVENT
        VAR_INPUT
          Robot_SetStartParam_IN : WORD;
        END_VAR
        SOCKETS
          AIAS_Skill : IAS_Skill;
        END_SOCKETS
      END_SUBAPPLICATION
      EVENT_CONNECTIONS
        DepotSkill.TurntablePresetPositionUpd TO TurntableSkill.Table_SetStartParam_REQ;
        START.COLD TO StorageSkill.INIT;
        START.WARM TO StorageSkill.INIT;
        StorageSkill.INITO TO TurntableSkill.INIT;
        TurntableSkill.INITO TO GripperSkill.INIT;
        START.COLD TO DepotSkill.INIT;
        START.WARM TO DepotSkill.INIT;
        DepotSkill.INITO TO HandlingSkill.INIT;
        HandlingSkill.RobotPositionUpd TO RobotSkill.SetStartParam_REQ;
        GripperSkill.INITO TO RobotSkill.INIT;
      END_CONNECTIONS
      DATA_CONNECTIONS
        DepotSkill.TurntablePresetPosition TO TurntableSkill.Table_SetStartParam_IN;
        HandlingSkill.RobotPresetPosition TO RobotSkill.Robot_SetStartParam_IN;
      END_CONNECTIONS
      ADAPTER_CONNECTIONS
        DepotSkill.AIAS_Skill_Storage TO StorageSkill.AIAS_Skill;
        DepotSkill.AIAS_Skill_Turntable TO TurntableSkill.AIAS_Skill;
        HandlingSkill.AIAS_Skill_Gripper TO GripperSkill.AIAS_Skill;
        Station1Control.ADepot TO DepotSkill.AIAS_Skill;
        Station1Control.AHandling TO HandlingSkill.AIAS_Skill;
        HandlingSkill.AIAS_Skill_Robot TO RobotSkill.AIAS_Skill;
      END_CONNECTIONS
    END_RESOURCE
    RESOURCE decentral : EMB_RES
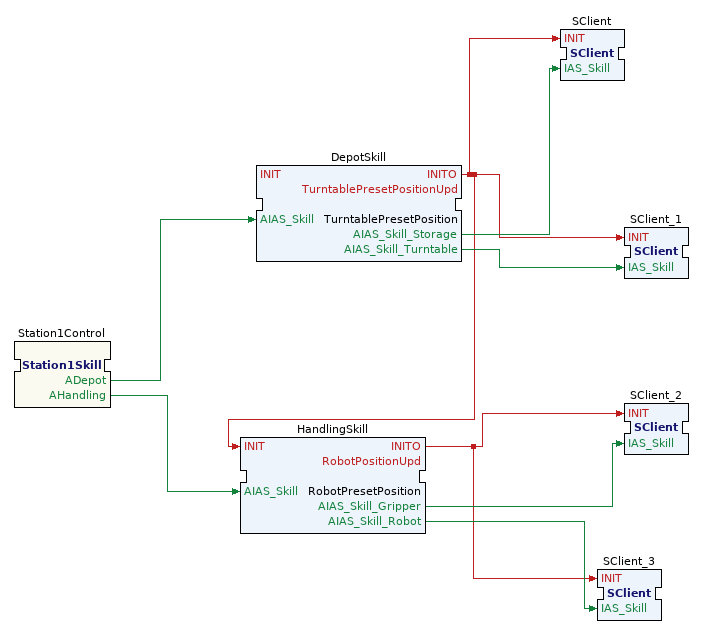
      FBS
        Station1Control : Station1Skill;
      END_FBS
      SUBAPPS
        SClient_2 : SClient;
        SClient_1 : SClient;
        SClient : SClient;
        SClient_3 : SClient;
      END_SUBAPPS
      SUBAPPLICATION HandlingSkill
        EVENT_INPUT
          INIT;
        END_EVENT
        EVENT_OUTPUT
          INITO;
          RobotPositionUpd;
        END_EVENT
        VAR_OUTPUT
          RobotPresetPosition : WORD;
        END_VAR
        SOCKETS
          AIAS_Skill : IAS_Skill;
        END_SOCKETS
        PLUGS
          AIAS_Skill_Gripper : IAS_Skill;
          AIAS_Skill_Robot : IAS_Skill;
        END_PLUGS
      END_SUBAPPLICATION
      SUBAPPLICATION DepotSkill
        EVENT_INPUT
          INIT;
        END_EVENT
        EVENT_OUTPUT
          INITO;
          TurntablePresetPositionUpd;
        END_EVENT
        VAR_OUTPUT
          TurntablePresetPosition : WORD;
        END_VAR
        SOCKETS
          AIAS_Skill : IAS_Skill;
        END_SOCKETS
        PLUGS
          AIAS_Skill_Storage : IAS_Skill;
          AIAS_Skill_Turntable : IAS_Skill;
        END_PLUGS
      END_SUBAPPLICATION
      EVENT_CONNECTIONS
        DepotSkill.INITO TO HandlingSkill.INIT;
        HandlingSkill.INITO TO SClient_3.INIT;
        HandlingSkill.INITO TO SClient_2.INIT;
        DepotSkill.INITO TO SClient_1.INIT;
        DepotSkill.INITO TO SClient.INIT;
      END_CONNECTIONS
      ADAPTER_CONNECTIONS
        Station1Control.ADepot TO DepotSkill.AIAS_Skill;
        Station1Control.AHandling TO HandlingSkill.AIAS_Skill;
        HandlingSkill.AIAS_Skill_Gripper TO SClient_2.IAS_Skill;
        DepotSkill.AIAS_Skill_Turntable TO SClient_1.IAS_Skill;
        DepotSkill.AIAS_Skill_Storage TO SClient.IAS_Skill;
        HandlingSkill.AIAS_Skill_Robot TO SClient_3.IAS_Skill;
      END_CONNECTIONS
    END_RESOURCE
  END_DEVICE
  DEVICE codeGenControl : FORTE_PC(MGR_ID := "localhost:61506")
    {SET_ATTRIBUTE(Profile, HOLOBLOC)} (* device profile *)
    RESOURCE central : EMB_RES
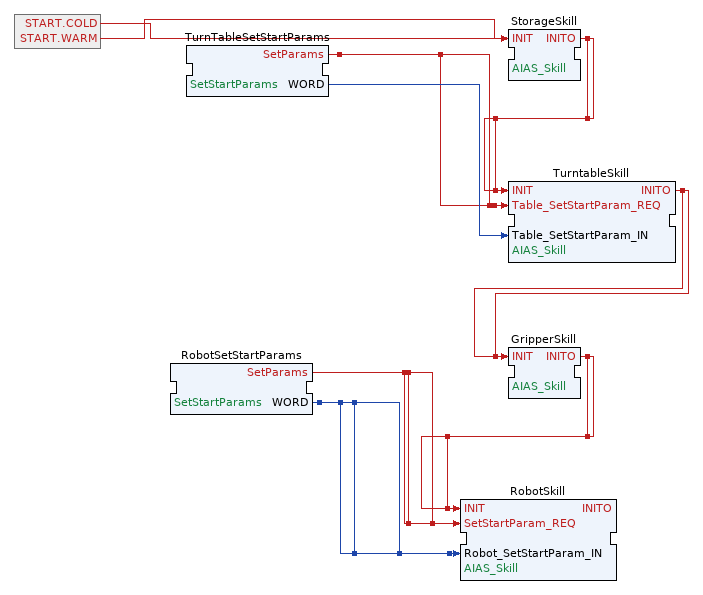
      SUBAPPLICATION RobotSetStartParams
        EVENT_OUTPUT
          SetParams;
        END_EVENT
        VAR_OUTPUT
          WORD : WORD;
        END_VAR
        SOCKETS
          SetStartParams : SetParams1Word;
        END_SOCKETS
      END_SUBAPPLICATION
      SUBAPPLICATION TurnTableSetStartParams
        EVENT_OUTPUT
          SetParams;
        END_EVENT
        VAR_OUTPUT
          WORD : WORD;
        END_VAR
        SOCKETS
          SetStartParams : SetParams1Word;
        END_SOCKETS
      END_SUBAPPLICATION
      SUBAPPLICATION StorageSkill
        EVENT_INPUT
          INIT;
        END_EVENT
        EVENT_OUTPUT
          INITO;
        END_EVENT
        SOCKETS
          AIAS_Skill : IAS_Skill;
        END_SOCKETS
      END_SUBAPPLICATION
      SUBAPPLICATION RobotSkill
        EVENT_INPUT
          INIT;
          SetStartParam_REQ;
        END_EVENT
        EVENT_OUTPUT
          INITO;
        END_EVENT
        VAR_INPUT
          Robot_SetStartParam_IN : WORD;
        END_VAR
        SOCKETS
          AIAS_Skill : IAS_Skill;
        END_SOCKETS
      END_SUBAPPLICATION
      SUBAPPLICATION TurntableSkill
        EVENT_INPUT
          INIT;
          Table_SetStartParam_REQ;
        END_EVENT
        EVENT_OUTPUT
          INITO;
        END_EVENT
        VAR_INPUT
          Table_SetStartParam_IN : WORD;
        END_VAR
        SOCKETS
          AIAS_Skill : IAS_Skill;
        END_SOCKETS
      END_SUBAPPLICATION
      SUBAPPLICATION GripperSkill
        EVENT_INPUT
          INIT;
        END_EVENT
        EVENT_OUTPUT
          INITO;
        END_EVENT
        SOCKETS
          AIAS_Skill : IAS_Skill;
        END_SOCKETS
      END_SUBAPPLICATION
      SUBAPPLICATION StorageSkill
        EVENT_INPUT
          INIT;
        END_EVENT
        EVENT_OUTPUT
          INITO;
        END_EVENT
        SOCKETS
          AIAS_Skill : IAS_Skill;
        END_SOCKETS
      END_SUBAPPLICATION
      SUBAPPLICATION TurntableSkill
        EVENT_INPUT
          INIT;
          Table_SetStartParam_REQ;
        END_EVENT
        EVENT_OUTPUT
          INITO;
        END_EVENT
        VAR_INPUT
          Table_SetStartParam_IN : WORD;
        END_VAR
        SOCKETS
          AIAS_Skill : IAS_Skill;
        END_SOCKETS
      END_SUBAPPLICATION
      SUBAPPLICATION GripperSkill
        EVENT_INPUT
          INIT;
        END_EVENT
        EVENT_OUTPUT
          INITO;
        END_EVENT
        SOCKETS
          AIAS_Skill : IAS_Skill;
        END_SOCKETS
      END_SUBAPPLICATION
      SUBAPPLICATION RobotSkill
        EVENT_INPUT
          INIT;
          SetStartParam_REQ;
        END_EVENT
        EVENT_OUTPUT
          INITO;
        END_EVENT
        VAR_INPUT
          Robot_SetStartParam_IN : WORD;
        END_VAR
        SOCKETS
          AIAS_Skill : IAS_Skill;
        END_SOCKETS
      END_SUBAPPLICATION
      SUBAPPLICATION TurnTableSetStartParams
        EVENT_OUTPUT
          SetParams;
        END_EVENT
        VAR_OUTPUT
          WORD : WORD;
        END_VAR
        SOCKETS
          SetStartParams : SetParams1Word;
        END_SOCKETS
      END_SUBAPPLICATION
      SUBAPPLICATION RobotSetStartParams
        EVENT_OUTPUT
          SetParams;
        END_EVENT
        VAR_OUTPUT
          WORD : WORD;
        END_VAR
        SOCKETS
          SetStartParams : SetParams1Word;
        END_SOCKETS
      END_SUBAPPLICATION
      SUBAPPLICATION TurntableSkill
        EVENT_INPUT
          INIT;
          Table_SetStartParam_REQ;
        END_EVENT
        EVENT_OUTPUT
          INITO;
        END_EVENT
        VAR_INPUT
          Table_SetStartParam_IN : WORD;
        END_VAR
        SOCKETS
          AIAS_Skill : IAS_Skill;
        END_SOCKETS
      END_SUBAPPLICATION
      SUBAPPLICATION GripperSkill
        EVENT_INPUT
          INIT;
        END_EVENT
        EVENT_OUTPUT
          INITO;
        END_EVENT
        SOCKETS
          AIAS_Skill : IAS_Skill;
        END_SOCKETS
      END_SUBAPPLICATION
      SUBAPPLICATION RobotSkill
        EVENT_INPUT
          INIT;
          SetStartParam_REQ;
        END_EVENT
        EVENT_OUTPUT
          INITO;
        END_EVENT
        VAR_INPUT
          Robot_SetStartParam_IN : WORD;
        END_VAR
        SOCKETS
          AIAS_Skill : IAS_Skill;
        END_SOCKETS
      END_SUBAPPLICATION
      SUBAPPLICATION StorageSkill
        EVENT_INPUT
          INIT;
        END_EVENT
        EVENT_OUTPUT
          INITO;
        END_EVENT
        SOCKETS
          AIAS_Skill : IAS_Skill;
        END_SOCKETS
      END_SUBAPPLICATION
      EVENT_CONNECTIONS
        RobotSetStartParams.SetParams TO RobotSkill.SetStartParam_REQ;
        StorageSkill.INITO TO TurntableSkill.INIT;
        TurnTableSetStartParams.SetParams TO TurntableSkill.Table_SetStartParam_REQ;
        TurntableSkill.INITO TO GripperSkill.INIT;
        GripperSkill.INITO TO RobotSkill.INIT;
        START.COLD TO StorageSkill.INIT;
        START.WARM TO StorageSkill.INIT;
        StorageSkill.INITO TO TurntableSkill.INIT;
        TurntableSkill.INITO TO GripperSkill.INIT;
        GripperSkill.INITO TO RobotSkill.INIT;
        TurnTableSetStartParams.SetParams TO TurntableSkill.Table_SetStartParam_REQ;
        RobotSetStartParams.SetParams TO RobotSkill.SetStartParam_REQ;
        TurnTableSetStartParams.SetParams TO TurntableSkill.Table_SetStartParam_REQ;
        TurntableSkill.INITO TO GripperSkill.INIT;
        GripperSkill.INITO TO RobotSkill.INIT;
        RobotSetStartParams.SetParams TO RobotSkill.SetStartParam_REQ;
        StorageSkill.INITO TO TurntableSkill.INIT;
      END_CONNECTIONS
      DATA_CONNECTIONS
        RobotSetStartParams.WORD TO RobotSkill.Robot_SetStartParam_IN;
        TurnTableSetStartParams.WORD TO TurntableSkill.Table_SetStartParam_IN;
        TurnTableSetStartParams.WORD TO TurntableSkill.Table_SetStartParam_IN;
        RobotSetStartParams.WORD TO RobotSkill.Robot_SetStartParam_IN;
        TurnTableSetStartParams.WORD TO TurntableSkill.Table_SetStartParam_IN;
        RobotSetStartParams.WORD TO RobotSkill.Robot_SetStartParam_IN;
      END_CONNECTIONS
    END_RESOURCE
    RESOURCE decentral : EMB_RES
      FBS
        Orchestrator : orchestratorFB;
        CLIENT_0 : CLIENT_0(QI := 1, ID := "opc_ua[CALL_METHOD;opc.tcp://localhost:4840#;/Objects/StorageSkill/cleanUp,1:s=StorageSkill_cleanUp]");
        CLIENT_1 : CLIENT_0(QI := 1, ID := "opc_ua[CALL_METHOD;opc.tcp://localhost:4840#;/Objects/StorageSkill/lock,1:s=StorageSkill_lock]");
        CLIENT_2 : CLIENT_0(QI := 1, ID := "opc_ua[CALL_METHOD;opc.tcp://localhost:4840#;/Objects/StorageSkill/reset,1:s=StorageSkill_reset]");
        CLIENT_3 : CLIENT_0(QI := 1, ID := "opc_ua[CALL_METHOD;opc.tcp://localhost:4840#;/Objects/StorageSkill/start,1:s=StorageSkill_start]");
        CLIENT_4 : CLIENT_0(QI := 1, ID := "opc_ua[CALL_METHOD;opc.tcp://localhost:4840#;/Objects/StorageSkill/stop,1:s=StorageSkill_stop]");
        CLIENT_5 : CLIENT_0(QI := 1, ID := "opc_ua[CALL_METHOD;opc.tcp://localhost:4840#;/Objects/StorageSkill/suspend,1:s=StorageSkill_suspend]");
        CLIENT_6 : CLIENT_0(QI := 1, ID := "opc_ua[CALL_METHOD;opc.tcp://localhost:4840#;/Objects/StorageSkill/unsuspend,1:s=StorageSkill_unsuspend]");
        SUBSCRIBE_2 : SUBSCRIBE_2(QI := 1, ID := "opc_ua[SUBSCRIBE;opc.tcp://localhost:4840#;/Objects/StorageSkill/currentState;/Objects/StorageSkill/lastTransition]");
        SETPARAMS1WORD_DEMUX_GEN : SETPARAMS1WORD_DEMUX_GEN;
        IAS_SKILL_DEMUX_GEN_1 : IAS_SKILL_DEMUX_GEN;
        SETPARAMS1WORD_DEMUX_GEN_1 : SETPARAMS1WORD_DEMUX_GEN;
        IAS_SKILL_DEMUX_GEN_2 : IAS_SKILL_DEMUX_GEN;
        IAS_SKILL_DEMUX_GEN_3 : IAS_SKILL_DEMUX_GEN;
        IAS_SKILL_DEMUX_GEN : IAS_SKILL_DEMUX_GEN;
        SUBSCRIBE_5 : SUBSCRIBE_2(QI := 1, ID := opc_ua[SUBSCRIBE;opc.tcp://localhost:4840#;/Objects/GripperSkill/currentState;/Objects/GripperSkill/lastTransition]);
        CLIENT_25 : CLIENT_0(QI := 1, ID := opc_ua[CALL_METHOD;opc.tcp://localhost:4840#;/Objects/GripperSkill/reset,1:s=GripperSkill_reset]);
        CLIENT_23 : CLIENT_0(QI := 1, ID := opc_ua[CALL_METHOD;opc.tcp://localhost:4840#;/Objects/GripperSkill/cleanUp,1:s=GripperSkill_cleanUp]);
        CLIENT_28 : CLIENT_0(QI := 1, ID := opc_ua[CALL_METHOD;opc.tcp://localhost:4840#;/Objects/GripperSkill/suspend,1:s=GripperSkill_suspend]);
        CLIENT_26 : CLIENT_0(QI := 1, ID := opc_ua[CALL_METHOD;opc.tcp://localhost:4840#;/Objects/GripperSkill/start,1:s=GripperSkill_start]);
        CLIENT_24 : CLIENT_0(QI := 1, ID := opc_ua[CALL_METHOD;opc.tcp://localhost:4840#;/Objects/GripperSkill/lock,1:s=GripperSkill_lock]);
        CLIENT_27 : CLIENT_0(QI := 1, ID := opc_ua[CALL_METHOD;opc.tcp://localhost:4840#;/Objects/GripperSkill/stop,1:s=GripperSkill_stop]);
        CLIENT_29 : CLIENT_0(QI := 1, ID := opc_ua[CALL_METHOD;opc.tcp://localhost:4840#;/Objects/GripperSkill/unsuspend,1:s=GripperSkill_unsuspend]);
        CLIENT_21 : CLIENT_0(QI := 1, ID := opc_ua[CALL_METHOD;opc.tcp://localhost:4840#;/Objects/RobotSkill/suspend,1:s=RobotSkill_suspend]);
        CLIENT_18 : CLIENT_0(QI := 1, ID := opc_ua[CALL_METHOD;opc.tcp://localhost:4840#;/Objects/RobotSkill/reset,1:s=RobotSkill_reset]);
        CLIENT_20 : CLIENT_0(QI := 1, ID := opc_ua[CALL_METHOD;opc.tcp://localhost:4840#;/Objects/RobotSkill/stop,1:s=RobotSkill_stop]);
        CLIENT_19 : CLIENT_0(QI := 1, ID := opc_ua[CALL_METHOD;opc.tcp://localhost:4840#;/Objects/RobotSkill/start,1:s=RobotSkill_start]);
        CLIENT_17 : CLIENT_0(QI := 1, ID := opc_ua[CALL_METHOD;opc.tcp://localhost:4840#;/Objects/RobotSkill/lock,1:s=RobotSkill_lock]);
        CLIENT_22 : CLIENT_0(QI := 1, ID := opc_ua[CALL_METHOD;opc.tcp://localhost:4840#;/Objects/RobotSkill/unsuspend,1:s=RobotSkill_unsuspend]);
        CLIENT_16 : CLIENT_0(QI := 1, ID := opc_ua[CALL_METHOD;opc.tcp://localhost:4840#;/Objects/RobotSkill/cleanUp,1:s=RobotSkill_cleanUp]);
        CLIENT_15 : CLIENT_1_0(QI := 1, ID := opc_ua[CALL_METHOD;opc.tcp://localhost:4840#;/Objects/RobotSetStartParams/IND,1:s=RobotSetStartParams_IND]);
        SUBSCRIBE_4 : SUBSCRIBE_2(QI := 1, ID := opc_ua[SUBSCRIBE;opc.tcp://localhost:4840#;/Objects/RobotSkill/currentState;/Objects/RobotSkill/lastTransition]);
        CLIENT_12 : CLIENT_0(QI := 1, ID := opc_ua[CALL_METHOD;opc.tcp://localhost:4840#;/Objects/TurntableSkill/stop,1:s=TurntableSkill_stop]);
        CLIENT_11 : CLIENT_0(QI := 1, ID := opc_ua[CALL_METHOD;opc.tcp://localhost:4840#;/Objects/TurntableSkill/start,1:s=TurntableSkill_start]);
        CLIENT_10 : CLIENT_0(QI := 1, ID := opc_ua[CALL_METHOD;opc.tcp://localhost:4840#;/Objects/TurntableSkill/reset,1:s=TurntableSkill_reset]);
        CLIENT_13 : CLIENT_0(QI := 1, ID := opc_ua[CALL_METHOD;opc.tcp://localhost:4840#;/Objects/TurntableSkill/suspend,1:s=TurntableSkill_suspend]);
        CLIENT_9 : CLIENT_0(QI := 1, ID := opc_ua[CALL_METHOD;opc.tcp://localhost:4840#;/Objects/TurntableSkill/lock,1:s=TurntableSkill_lock]);
        CLIENT_8 : CLIENT_0(QI := 1, ID := opc_ua[CALL_METHOD;opc.tcp://localhost:4840#;/Objects/TurntableSkill/cleanUp,1:s=TurntableSkill_cleanUp]);
        CLIENT_14 : CLIENT_0(QI := 1, ID := opc_ua[CALL_METHOD;opc.tcp://localhost:4840#;/Objects/TurntableSkill/unsuspend,1:s=TurntableSkill_unsuspend]);
        CLIENT_7 : CLIENT_1_0(QI := 1, ID := opc_ua[CALL_METHOD;opc.tcp://localhost:4840#;/Objects/TurnTableSetStartParams/IND,1:s=TurnTableSetStartParams_IND]);
        SUBSCRIBE_3 : SUBSCRIBE_2(QI := 1, ID := opc_ua[SUBSCRIBE;opc.tcp://localhost:4840#;/Objects/TurntableSkill/currentState;/Objects/TurntableSkill/lastTransition]);
      END_FBS
      EVENT_CONNECTIONS
        Orchestrator.doRndCnt TO Orchestrator.rndCntDone;
        Orchestrator.doRepCnt TO Orchestrator.repCntDone;
        START.COLD TO SUBSCRIBE_2.INIT;
        START.WARM TO SUBSCRIBE_2.INIT;
        SUBSCRIBE_2.INITO TO CLIENT_0.INIT;
        CLIENT_0.INITO TO CLIENT_1.INIT;
        CLIENT_1.INITO TO CLIENT_2.INIT;
        CLIENT_2.INITO TO CLIENT_3.INIT;
        CLIENT_3.INITO TO CLIENT_4.INIT;
        CLIENT_4.INITO TO CLIENT_5.INIT;
        CLIENT_5.INITO TO CLIENT_6.INIT;
        IAS_SKILL_DEMUX_GEN.cleanUp TO CLIENT_0.REQ;
        IAS_SKILL_DEMUX_GEN.lock TO CLIENT_1.REQ;
        IAS_SKILL_DEMUX_GEN.reset TO CLIENT_2.REQ;
        IAS_SKILL_DEMUX_GEN.start TO CLIENT_3.REQ;
        IAS_SKILL_DEMUX_GEN.stop TO CLIENT_4.REQ;
        IAS_SKILL_DEMUX_GEN.suspend TO CLIENT_5.REQ;
        IAS_SKILL_DEMUX_GEN.unsuspend TO CLIENT_6.REQ;
        SUBSCRIBE_2.IND TO IAS_SKILL_DEMUX_GEN.RSP;
        SUBSCRIBE_5.IND TO IAS_SKILL_DEMUX_GEN_3.RSP;
        START.COLD TO SUBSCRIBE_5.INIT;
        START.WARM TO SUBSCRIBE_5.INIT;
        SUBSCRIBE_5.INITO TO CLIENT_23.INIT;
        IAS_SKILL_DEMUX_GEN_3.lock TO CLIENT_24.REQ;
        IAS_SKILL_DEMUX_GEN_3.suspend TO CLIENT_28.REQ;
        IAS_SKILL_DEMUX_GEN_3.cleanUp TO CLIENT_23.REQ;
        CLIENT_28.INITO TO CLIENT_29.INIT;
        IAS_SKILL_DEMUX_GEN_3.unsuspend TO CLIENT_29.REQ;
        CLIENT_25.INITO TO CLIENT_26.INIT;
        CLIENT_27.INITO TO CLIENT_28.INIT;
        IAS_SKILL_DEMUX_GEN_3.start TO CLIENT_26.REQ;
        CLIENT_24.INITO TO CLIENT_25.INIT;
        CLIENT_23.INITO TO CLIENT_24.INIT;
        CLIENT_26.INITO TO CLIENT_27.INIT;
        IAS_SKILL_DEMUX_GEN_3.reset TO CLIENT_25.REQ;
        IAS_SKILL_DEMUX_GEN_3.stop TO CLIENT_27.REQ;
        IAS_SKILL_DEMUX_GEN_2.suspend TO CLIENT_21.REQ;
        IAS_SKILL_DEMUX_GEN_2.reset TO CLIENT_18.REQ;
        IAS_SKILL_DEMUX_GEN_2.stop TO CLIENT_20.REQ;
        IAS_SKILL_DEMUX_GEN_2.start TO CLIENT_19.REQ;
        IAS_SKILL_DEMUX_GEN_2.lock TO CLIENT_17.REQ;
        IAS_SKILL_DEMUX_GEN_2.unsuspend TO CLIENT_22.REQ;
        IAS_SKILL_DEMUX_GEN_2.cleanUp TO CLIENT_16.REQ;
        CLIENT_17.INITO TO CLIENT_18.INIT;
        CLIENT_21.INITO TO CLIENT_22.INIT;
        CLIENT_18.INITO TO CLIENT_19.INIT;
        CLIENT_16.INITO TO CLIENT_17.INIT;
        CLIENT_20.INITO TO CLIENT_21.INIT;
        CLIENT_19.INITO TO CLIENT_20.INIT;
        SETPARAMS1WORD_DEMUX_GEN_1.IND TO CLIENT_15.REQ;
        START.COLD TO CLIENT_15.INIT;
        START.WARM TO CLIENT_15.INIT;
        SUBSCRIBE_4.IND TO IAS_SKILL_DEMUX_GEN_2.RSP;
        SUBSCRIBE_4.INITO TO CLIENT_16.INIT;
        START.COLD TO SUBSCRIBE_4.INIT;
        START.WARM TO SUBSCRIBE_4.INIT;
        IAS_SKILL_DEMUX_GEN_1.stop TO CLIENT_12.REQ;
        IAS_SKILL_DEMUX_GEN_1.start TO CLIENT_11.REQ;
        IAS_SKILL_DEMUX_GEN_1.reset TO CLIENT_10.REQ;
        IAS_SKILL_DEMUX_GEN_1.suspend TO CLIENT_13.REQ;
        IAS_SKILL_DEMUX_GEN_1.lock TO CLIENT_9.REQ;
        IAS_SKILL_DEMUX_GEN_1.cleanUp TO CLIENT_8.REQ;
        IAS_SKILL_DEMUX_GEN_1.unsuspend TO CLIENT_14.REQ;
        CLIENT_10.INITO TO CLIENT_11.INIT;
        CLIENT_9.INITO TO CLIENT_10.INIT;
        CLIENT_13.INITO TO CLIENT_14.INIT;
        CLIENT_8.INITO TO CLIENT_9.INIT;
        CLIENT_11.INITO TO CLIENT_12.INIT;
        CLIENT_12.INITO TO CLIENT_13.INIT;
        SETPARAMS1WORD_DEMUX_GEN.IND TO CLIENT_7.REQ;
        START.COLD TO CLIENT_7.INIT;
        START.WARM TO CLIENT_7.INIT;
        SUBSCRIBE_3.IND TO IAS_SKILL_DEMUX_GEN_1.RSP;
        SUBSCRIBE_3.INITO TO CLIENT_8.INIT;
        START.COLD TO SUBSCRIBE_3.INIT;
        START.WARM TO SUBSCRIBE_3.INIT;
      END_CONNECTIONS
      DATA_CONNECTIONS
        SUBSCRIBE_2.RD_1 TO IAS_SKILL_DEMUX_GEN.currentState;
        SUBSCRIBE_2.RD_2 TO IAS_SKILL_DEMUX_GEN.lastTransition;
        SUBSCRIBE_5.RD_2 TO IAS_SKILL_DEMUX_GEN_3.lastTransition;
        SUBSCRIBE_5.RD_1 TO IAS_SKILL_DEMUX_GEN_3.currentState;
        SETPARAMS1WORD_DEMUX_GEN_1.DATA TO CLIENT_15.SD_1;
        SUBSCRIBE_4.RD_2 TO IAS_SKILL_DEMUX_GEN_2.lastTransition;
        SUBSCRIBE_4.RD_1 TO IAS_SKILL_DEMUX_GEN_2.currentState;
        SETPARAMS1WORD_DEMUX_GEN.DATA TO CLIENT_7.SD_1;
        SUBSCRIBE_3.RD_2 TO IAS_SKILL_DEMUX_GEN_1.lastTransition;
        SUBSCRIBE_3.RD_1 TO IAS_SKILL_DEMUX_GEN_1.currentState;
      END_CONNECTIONS
      ADAPTER_CONNECTIONS
        Orchestrator.TurnTableSetStartParams_SetParams1Word TO SETPARAMS1WORD_DEMUX_GEN.SetParams1Word;
        Orchestrator.TurntableSkill_IAS_Skill TO IAS_SKILL_DEMUX_GEN_1.IAS_Skill;
        Orchestrator.RobotSetStartParams_SetParams1Word TO SETPARAMS1WORD_DEMUX_GEN_1.SetParams1Word;
        Orchestrator.RobotSkill_IAS_Skill TO IAS_SKILL_DEMUX_GEN_2.IAS_Skill;
        Orchestrator.GripperSkill_IAS_Skill TO IAS_SKILL_DEMUX_GEN_3.IAS_Skill;
        Orchestrator.StorageSkill_IAS_Skill TO IAS_SKILL_DEMUX_GEN.IAS_Skill;
      END_CONNECTIONS
    END_RESOURCE
  END_DEVICE
  DEVICE deviceAdapter : FORTE_PC(MGR_ID := "localhost:61507")
    {SET_ATTRIBUTE(Profile, HOLOBLOC)} (* device profile *)
    RESOURCE EMB_RES : EMB_RES
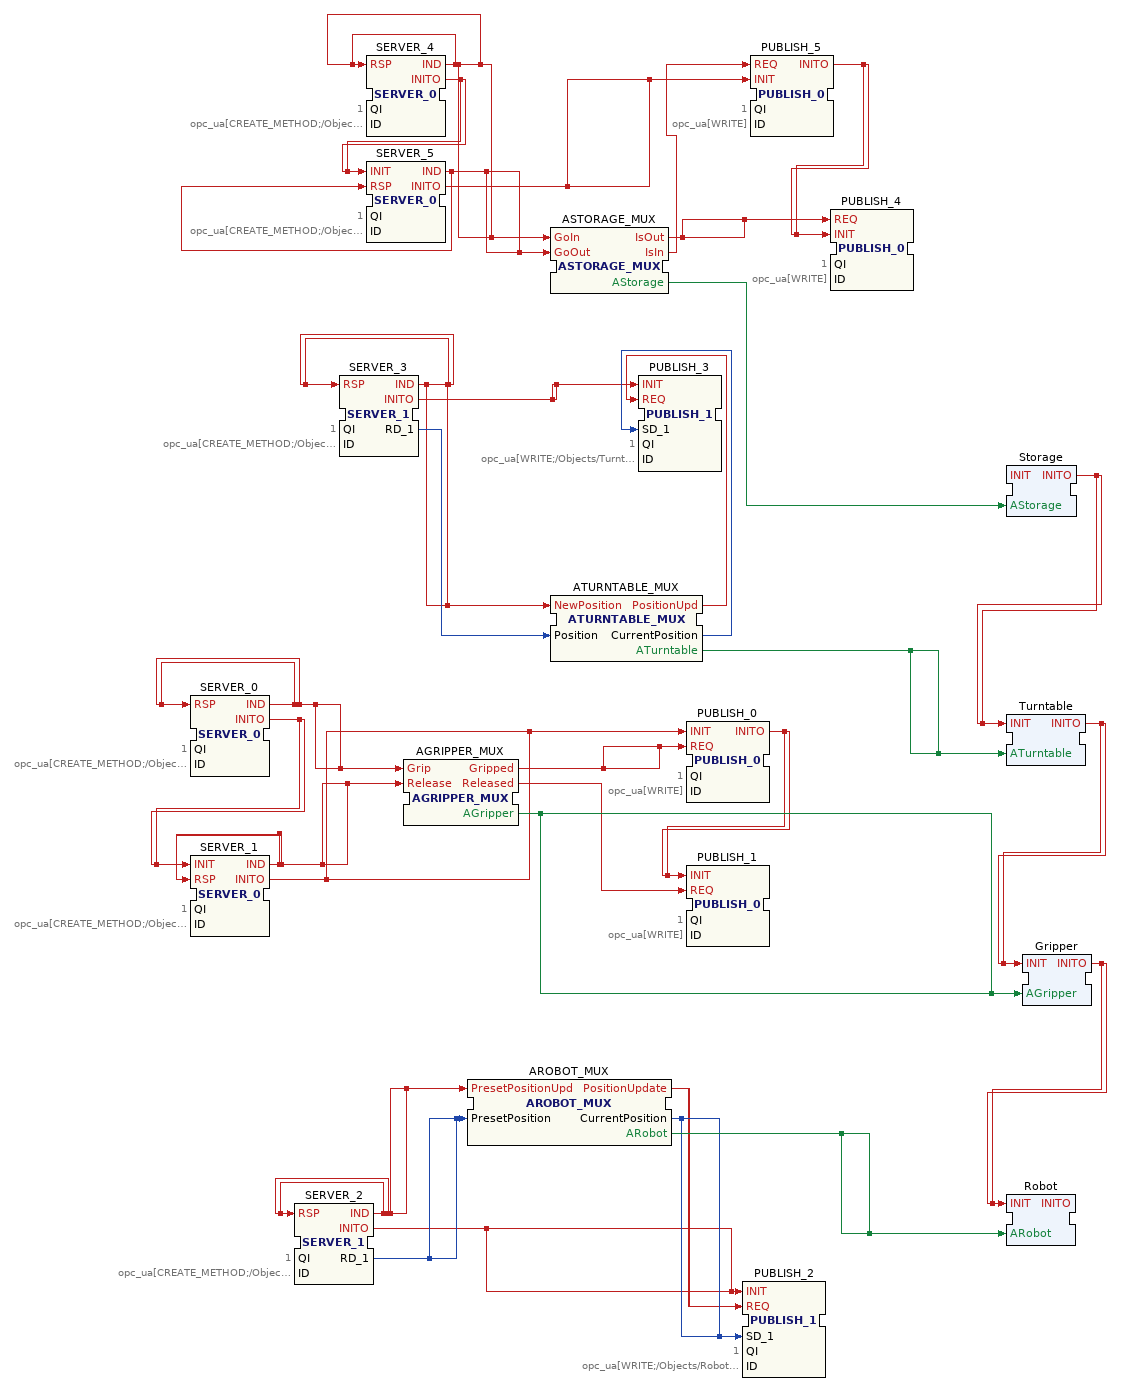
      FBS
        SERVER_0 : SERVER_0(QI := 1, ID := opc_ua[CREATE_METHOD;/Objects/Gripper/Grip,1:s=Gripper_Grip]);
        PUBLISH_0 : PUBLISH_0(QI := 1, ID := opc_ua[WRITE]);
        SERVER_1 : SERVER_0(QI := 1, ID := opc_ua[CREATE_METHOD;/Objects/Gripper/Release,1:s=Gripper_Release]);
        PUBLISH_1 : PUBLISH_0(QI := 1, ID := opc_ua[WRITE]);
        AGRIPPER_MUX : AGRIPPER_MUX;
        SERVER_2 : SERVER_1(QI := 1, ID := opc_ua[CREATE_METHOD;/Objects/Robot/PresetPositionUpd,1:s=Robot_PresetPositionUpd]);
        AROBOT_MUX : AROBOT_MUX;
        PUBLISH_2 : PUBLISH_1(QI := 1, ID := opc_ua[WRITE;/Objects/Robot/CurrentPosition]);
        PUBLISH_3 : PUBLISH_1(QI := 1, ID := opc_ua[WRITE;/Objects/Turntable/CurrentPosition]);
        SERVER_3 : SERVER_1(QI := 1, ID := opc_ua[CREATE_METHOD;/Objects/Turntable/NewPosition,1:s=Turntable_NewPosition]);
        ATURNTABLE_MUX : ATURNTABLE_MUX;
        PUBLISH_4 : PUBLISH_0(QI := 1, ID := opc_ua[WRITE]);
        ASTORAGE_MUX : ASTORAGE_MUX;
        PUBLISH_5 : PUBLISH_0(QI := 1, ID := opc_ua[WRITE]);
        SERVER_4 : SERVER_0(QI := 1, ID := opc_ua[CREATE_METHOD;/Objects/Storage/GoIn,1:s=Storage_GoIn]);
        SERVER_5 : SERVER_0(QI := 1, ID := opc_ua[CREATE_METHOD;/Objects/Storage/GoOut,1:s=Storage_GoOut]);
      END_FBS
      SUBAPPLICATION Robot
        EVENT_INPUT
          INIT;
        END_EVENT
        EVENT_OUTPUT
          INITO;
        END_EVENT
        SOCKETS
          ARobot : ARobot;
        END_SOCKETS
      END_SUBAPPLICATION
      SUBAPPLICATION Gripper
        EVENT_INPUT
          INIT;
        END_EVENT
        EVENT_OUTPUT
          INITO;
        END_EVENT
        SOCKETS
          AGripper : AGripper;
        END_SOCKETS
      END_SUBAPPLICATION
      SUBAPPLICATION Turntable
        EVENT_INPUT
          INIT;
        END_EVENT
        EVENT_OUTPUT
          INITO;
        END_EVENT
        SOCKETS
          ATurntable : ATurntable;
        END_SOCKETS
      END_SUBAPPLICATION
      SUBAPPLICATION Storage
        EVENT_INPUT
          INIT;
        END_EVENT
        EVENT_OUTPUT
          INITO;
        END_EVENT
        SOCKETS
          AStorage : AStorage;
        END_SOCKETS
      END_SUBAPPLICATION
      EVENT_CONNECTIONS
        Gripper.INITO TO Robot.INIT;
        Turntable.INITO TO Gripper.INIT;
        Storage.INITO TO Turntable.INIT;
        SERVER_0.IND TO SERVER_0.RSP;
        SERVER_0.INITO TO SERVER_1.INIT;
        SERVER_1.IND TO SERVER_1.RSP;
        SERVER_1.INITO TO PUBLISH_0.INIT;
        PUBLISH_0.INITO TO PUBLISH_1.INIT;
        SERVER_0.IND TO AGRIPPER_MUX.Grip;
        SERVER_1.IND TO AGRIPPER_MUX.Release;
        AGRIPPER_MUX.Gripped TO PUBLISH_0.REQ;
        AGRIPPER_MUX.Released TO PUBLISH_1.REQ;
        SERVER_2.IND TO SERVER_2.RSP;
        SERVER_2.IND TO AROBOT_MUX.PresetPositionUpd;
        SERVER_2.INITO TO PUBLISH_2.INIT;
        AROBOT_MUX.PositionUpdate TO PUBLISH_2.REQ;
        SERVER_3.IND TO SERVER_3.RSP;
        SERVER_3.INITO TO PUBLISH_3.INIT;
        SERVER_3.IND TO ATURNTABLE_MUX.NewPosition;
        ATURNTABLE_MUX.PositionUpd TO PUBLISH_3.REQ;
        ASTORAGE_MUX.IsOut TO PUBLISH_4.REQ;
        ASTORAGE_MUX.IsIn TO PUBLISH_5.REQ;
        PUBLISH_5.INITO TO PUBLISH_4.INIT;
        SERVER_4.IND TO SERVER_4.RSP;
        SERVER_4.IND TO ASTORAGE_MUX.GoIn;
        SERVER_4.INITO TO SERVER_5.INIT;
        SERVER_5.IND TO SERVER_5.RSP;
        SERVER_5.INITO TO PUBLISH_5.INIT;
        SERVER_5.IND TO ASTORAGE_MUX.GoOut;
        Gripper.INITO TO Robot.INIT;
        Turntable.INITO TO Gripper.INIT;
        Storage.INITO TO Turntable.INIT;
        SERVER_0.IND TO SERVER_0.RSP;
        SERVER_0.INITO TO SERVER_1.INIT;
        SERVER_1.IND TO SERVER_1.RSP;
        SERVER_1.INITO TO PUBLISH_0.INIT;
        PUBLISH_0.INITO TO PUBLISH_1.INIT;
        SERVER_0.IND TO AGRIPPER_MUX.Grip;
        SERVER_1.IND TO AGRIPPER_MUX.Release;
        AGRIPPER_MUX.Gripped TO PUBLISH_0.REQ;
        AGRIPPER_MUX.Released TO PUBLISH_1.REQ;
        SERVER_2.IND TO SERVER_2.RSP;
        SERVER_2.IND TO AROBOT_MUX.PresetPositionUpd;
        SERVER_2.INITO TO PUBLISH_2.INIT;
        AROBOT_MUX.PositionUpdate TO PUBLISH_2.REQ;
        SERVER_3.IND TO SERVER_3.RSP;
        SERVER_3.INITO TO PUBLISH_3.INIT;
        SERVER_3.IND TO ATURNTABLE_MUX.NewPosition;
        ATURNTABLE_MUX.PositionUpd TO PUBLISH_3.REQ;
        ASTORAGE_MUX.IsOut TO PUBLISH_4.REQ;
        ASTORAGE_MUX.IsIn TO PUBLISH_5.REQ;
        PUBLISH_5.INITO TO PUBLISH_4.INIT;
        SERVER_4.IND TO SERVER_4.RSP;
        SERVER_4.IND TO ASTORAGE_MUX.GoIn;
        SERVER_4.INITO TO SERVER_5.INIT;
        SERVER_5.IND TO SERVER_5.RSP;
        SERVER_5.INITO TO PUBLISH_5.INIT;
        SERVER_5.IND TO ASTORAGE_MUX.GoOut;
      END_CONNECTIONS
      DATA_CONNECTIONS
        SERVER_2.RD_1 TO AROBOT_MUX.PresetPosition;
        AROBOT_MUX.CurrentPosition TO PUBLISH_2.SD_1;
        SERVER_3.RD_1 TO ATURNTABLE_MUX.Position;
        ATURNTABLE_MUX.CurrentPosition TO PUBLISH_3.SD_1;
        SERVER_2.RD_1 TO AROBOT_MUX.PresetPosition;
        AROBOT_MUX.CurrentPosition TO PUBLISH_2.SD_1;
        SERVER_3.RD_1 TO ATURNTABLE_MUX.Position;
        ATURNTABLE_MUX.CurrentPosition TO PUBLISH_3.SD_1;
      END_CONNECTIONS
      ADAPTER_CONNECTIONS
        AGRIPPER_MUX.AGripper TO Gripper.AGripper;
        AROBOT_MUX.ARobot TO Robot.ARobot;
        ATURNTABLE_MUX.ATurntable TO Turntable.ATurntable;
        ASTORAGE_MUX.AStorage TO Storage.AStorage;
        AGRIPPER_MUX.AGripper TO Gripper.AGripper;
        AROBOT_MUX.ARobot TO Robot.ARobot;
        ATURNTABLE_MUX.ATurntable TO Turntable.ATurntable;
        ASTORAGE_MUX.AStorage TO Storage.AStorage;
      END_CONNECTIONS
    END_RESOURCE
  END_DEVICE
  DEVICE allDevicesOnOneForte : FORTE_PC(MGR_ID := "localhost:61510")
    {SET_ATTRIBUTE(Profile, HOLOBLOC)} (* device profile *)
    RESOURCE emulator : EMB_RES
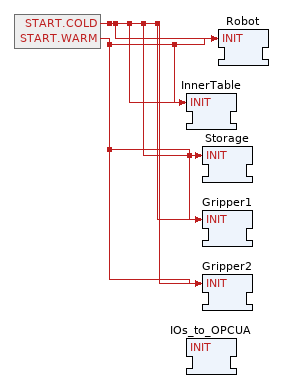
      SUBAPPLICATION Robot
        EVENT_INPUT
          INIT;
        END_EVENT
      END_SUBAPPLICATION
      SUBAPPLICATION Storage
        EVENT_INPUT
          INIT;
        END_EVENT
      END_SUBAPPLICATION
      SUBAPPLICATION InnerTable
        EVENT_INPUT
          INIT;
        END_EVENT
      END_SUBAPPLICATION
      SUBAPPLICATION Gripper1
        EVENT_INPUT
          INIT;
        END_EVENT
      END_SUBAPPLICATION
      SUBAPPLICATION Gripper2
        EVENT_INPUT
          INIT;
        END_EVENT
      END_SUBAPPLICATION
      SUBAPPLICATION IOs_to_OPCUA
        EVENT_INPUT
          INIT;
        END_EVENT
      END_SUBAPPLICATION
      EVENT_CONNECTIONS
        START.COLD TO Robot.INIT;
        START.WARM TO Robot.INIT;
        START.COLD TO InnerTable.INIT;
        START.WARM TO InnerTable.INIT;
        START.COLD TO Storage.INIT;
        START.WARM TO Storage.INIT;
        START.COLD TO Gripper1.INIT;
        START.WARM TO Gripper1.INIT;
        START.COLD TO Gripper2.INIT;
        START.WARM TO Gripper2.INIT;
      END_CONNECTIONS
    END_RESOURCE
    RESOURCE hier_decentral : EMB_RES
      FBS
        AROBOT_MUX : AROBOT_MUX;
        SERVER_2 : SERVER_0_1(QI := 1, ID := opc_ua[CREATE_METHOD;/Objects/Robot/PresetPositionUpd]);
        PUBLISH_3 : PUBLISH_1(QI := 1, ID := opc_ua[WRITE;/Objects/Turntable/CurrentPosition]);
        SERVER_0 : SERVER_0(QI := 1, ID := opc_ua[CREATE_METHOD;/Objects/Gripper/Grip]);
        SERVER_3 : SERVER_0_1(QI := 1, ID := opc_ua[CREATE_METHOD;/Objects/Turntable/NewPosition]);
        AGRIPPER_MUX : AGRIPPER_MUX;
        ATURNTABLE_MUX : ATURNTABLE_MUX;
        PUBLISH_0 : PUBLISH_1(QI := 1, ID := opc_ua[WRITE;/Objects/Gripper/Gripped]);
        E_RS_2 : E_RS;
        PUBLISH_2 : PUBLISH_1(QI := 1, ID := opc_ua[WRITE;/Objects/Robot/CurrentPosition]);
        E_RS_3 : E_RS;
        PUBLISH_1 : PUBLISH_1(QI := 1, ID := opc_ua[WRITE;/Objects/Gripper/Released]);
        SERVER_1 : SERVER_0(QI := 1, ID := opc_ua[CREATE_METHOD;/Objects/Gripper/Release]);
        SERVER_5 : SERVER_0(QI := 1, ID := opc_ua[CREATE_METHOD;/Objects/Storage/GoOut,1:s=Storage_GoOut]);
        E_RS : E_RS;
        ASTORAGE_MUX : ASTORAGE_MUX;
        SERVER_4 : SERVER_0(QI := 1, ID := opc_ua[CREATE_METHOD;/Objects/Storage/GoIn,1:s=Storage_GoIn]);
        PUBLISH_4 : PUBLISH_1(QI := 1, ID := opc_ua[WRITE;/Objects/Storage/IsOut]);
        E_RS_1 : E_RS;
        PUBLISH_5 : PUBLISH_1(QI := 1, ID := opc_ua[WRITE;/Objects/Storage/IsIn]);
        CLIENT_5 : CLIENT_0(QI := 1, ID := opc_ua[CALL_METHOD;opc.tcp://localhost:4850#;/Objects/Gripper/Release]);
        CLIENT_1 : CLIENT_1_0(QI := 1, ID := opc_ua[CALL_METHOD;opc.tcp://localhost:4850#;/Objects/Robot/PresetPositionUpd]);
        SUBSCRIBE_1 : SUBSCRIBE_1(QI := 1, ID := opc_ua[SUBSCRIBE;opc.tcp://localhost:4850#;/Objects/Robot/CurrentPosition]);
        CLIENT_4 : CLIENT_0(QI := 1, ID := opc_ua[CALL_METHOD;opc.tcp://localhost:4850#;/Objects/Gripper/Grip]);
        SUBSCRIBE_0 : SUBSCRIBE_0(QI := 1, ID := opc_ua[SUBSCRIBE;opc.tcp://localhost:4840#]);
        AGRIPPER_DEMUX : AGRIPPER_DEMUX;
        HandlingControl : HandlingControl;
        SUBSCRIBE_3 : SUBSCRIBE_1(QI := 1, ID := opc_ua[SUBSCRIBE;opc.tcp://localhost:4850#;/Objects/Storage/IsOut]);
        SUBSCRIBE_9 : SUBSCRIBE_1(QI := 1, ID := opc_ua[SUBSCRIBE;opc.tcp://localhost:4850#;/Objects/Storage/IsIn]);
        E_SWITCH_3 : E_SWITCH;
        DepotControl : DepotControl;
        ATURNTABLE_DEMUX : ATURNTABLE_DEMUX;
        E_SWITCH_1 : E_SWITCH;
        CLIENT_2 : CLIENT_1_0(QI := 1, ID := opc_ua[CALL_METHOD;opc.tcp://localhost:4850#;/Objects/Turntable/NewPosition]);
        E_SWITCH_2 : E_SWITCH;
        AROBOT_DEMUX : AROBOT_DEMUX;
        ASTORAGE_DEMUX : ASTORAGE_DEMUX;
        SUBSCRIBE_5 : SUBSCRIBE_1(QI := 1, ID := opc_ua[SUBSCRIBE;opc.tcp://localhost:4850#;/Objects/Gripper/Released]);
        Station1Control : Station1Control;
        CLIENT_3 : CLIENT_0(QI := 1, ID := opc_ua[CALL_METHOD;opc.tcp://localhost:4850#;/Objects/Storage/GoOut]);
        CLIENT_0 : CLIENT_0(QI := 1, ID := opc_ua[CALL_METHOD;opc.tcp://localhost:4850#;/Objects/Storage/GoIn]);
        SUBSCRIBE_2 : SUBSCRIBE_1(QI := 1, ID := opc_ua[SUBSCRIBE;opc.tcp://localhost:4850#;/Objects/Turntable/CurrentPosition]);
        E_SWITCH : E_SWITCH;
        SUBSCRIBE_4 : SUBSCRIBE_1(QI := 1, ID := opc_ua[SUBSCRIBE;opc.tcp://localhost:4850#;/Objects/Gripper/Gripped]);
      END_FBS
      SUBAPPLICATION Robot
        EVENT_INPUT
          INIT;
        END_EVENT
        EVENT_OUTPUT
          INITO;
        END_EVENT
        SOCKETS
          ARobot : ARobot;
        END_SOCKETS
      END_SUBAPPLICATION
      SUBAPPLICATION Turntable
        EVENT_INPUT
          INIT;
        END_EVENT
        EVENT_OUTPUT
          INITO;
        END_EVENT
        SOCKETS
          ATurntable : ATurntable;
        END_SOCKETS
      END_SUBAPPLICATION
      SUBAPPLICATION Gripper
        EVENT_INPUT
          INIT;
        END_EVENT
        EVENT_OUTPUT
          INITO;
        END_EVENT
        SOCKETS
          AGripper : AGripper;
        END_SOCKETS
      END_SUBAPPLICATION
      SUBAPPLICATION Storage
        EVENT_INPUT
          INIT;
        END_EVENT
        EVENT_OUTPUT
          INITO;
        END_EVENT
        SOCKETS
          AStorage : AStorage;
        END_SOCKETS
      END_SUBAPPLICATION
      EVENT_CONNECTIONS
        SERVER_2.IND TO SERVER_2.RSP;
        SERVER_2.IND TO AROBOT_MUX.PresetPositionUpd;
        SERVER_0.IND TO SERVER_0.RSP;
        SERVER_3.IND TO SERVER_3.RSP;
        SERVER_3.INITO TO PUBLISH_3.INIT;
        SERVER_0.IND TO AGRIPPER_MUX.Grip;
        Robot.INITO TO SERVER_2.INIT;
        SERVER_3.IND TO ATURNTABLE_MUX.NewPosition;
        ATURNTABLE_MUX.PositionUpd TO PUBLISH_3.REQ;
        Turntable.INITO TO SERVER_3.INIT;
        AGRIPPER_MUX.Released TO E_RS_2.R;
        AGRIPPER_MUX.Gripped TO E_RS_2.S;
        E_RS_2.EO TO PUBLISH_0.REQ;
        Turntable.INITO TO Gripper.INIT;
        Gripper.INITO TO Robot.INIT;
        Gripper.INITO TO SERVER_0.INIT;
        SERVER_2.INITO TO PUBLISH_2.INIT;
        AROBOT_MUX.PositionUpdate TO PUBLISH_2.REQ;
        AGRIPPER_MUX.Gripped TO E_RS_3.R;
        AGRIPPER_MUX.Released TO E_RS_3.S;
        PUBLISH_0.INITO TO PUBLISH_1.INIT;
        E_RS_3.EO TO PUBLISH_1.REQ;
        SERVER_0.INITO TO SERVER_1.INIT;
        SERVER_1.IND TO SERVER_1.RSP;
        SERVER_1.INITO TO PUBLISH_0.INIT;
        SERVER_1.IND TO AGRIPPER_MUX.Release;
        SERVER_5.IND TO SERVER_5.RSP;
        SERVER_5.IND TO ASTORAGE_MUX.GoOut;
        ASTORAGE_MUX.IsIn TO E_RS.R;
        ASTORAGE_MUX.IsOut TO E_RS.S;
        SERVER_4.IND TO SERVER_4.RSP;
        SERVER_4.INITO TO SERVER_5.INIT;
        SERVER_4.IND TO ASTORAGE_MUX.GoIn;
        E_RS.EO TO PUBLISH_4.REQ;
        SERVER_5.INITO TO Storage.INIT;
        Storage.INITO TO Turntable.INIT;
        ASTORAGE_MUX.IsOut TO E_RS_1.R;
        ASTORAGE_MUX.IsIn TO E_RS_1.S;
        SERVER_5.INITO TO PUBLISH_5.INIT;
        E_RS_1.EO TO PUBLISH_5.REQ;
        PUBLISH_5.INITO TO PUBLISH_4.INIT;
        SUBSCRIBE_1.INITO TO CLIENT_1.INIT;
        CLIENT_4.INITO TO CLIENT_5.INIT;
        AGRIPPER_DEMUX.Grip TO CLIENT_4.REQ;
        AGRIPPER_DEMUX.Release TO CLIENT_5.REQ;
        SUBSCRIBE_9.INITO TO SUBSCRIBE_3.INIT;
        AGRIPPER_DEMUX.Release TO E_SWITCH_3.EI;
        E_SWITCH_3.EO1 TO AGRIPPER_DEMUX.Released;
        SUBSCRIBE_9.IND TO E_SWITCH_1.EI;
        ATURNTABLE_DEMUX.NewPosition TO CLIENT_2.REQ;
        AGRIPPER_DEMUX.Grip TO E_SWITCH_2.EI;
        E_SWITCH_2.EO1 TO AGRIPPER_DEMUX.Gripped;
        SUBSCRIBE_1.IND TO AROBOT_DEMUX.PositionUpdate;
        AROBOT_DEMUX.PresetPositionUpd TO CLIENT_1.REQ;
        E_SWITCH_1.EO1 TO ASTORAGE_DEMUX.IsIn;
        ASTORAGE_DEMUX.GoIn TO E_SWITCH_1.EI;
        SUBSCRIBE_5.INITO TO SUBSCRIBE_1.INIT;
        SUBSCRIBE_5.INITO TO CLIENT_4.INIT;
        SUBSCRIBE_5.IND TO E_SWITCH_3.EI;
        ASTORAGE_DEMUX.GoOut TO CLIENT_3.REQ;
        SUBSCRIBE_3.INITO TO CLIENT_0.INIT;
        ASTORAGE_DEMUX.GoIn TO CLIENT_0.REQ;
        CLIENT_0.INITO TO CLIENT_3.INIT;
        CLIENT_3.INITO TO SUBSCRIBE_2.INIT;
        SUBSCRIBE_2.INITO TO CLIENT_2.INIT;
        SUBSCRIBE_2.IND TO ATURNTABLE_DEMUX.PositionUpd;
        ASTORAGE_DEMUX.GoOut TO E_SWITCH.EI;
        SUBSCRIBE_3.IND TO E_SWITCH.EI;
        E_SWITCH.EO1 TO ASTORAGE_DEMUX.IsOut;
        SUBSCRIBE_2.INITO TO SUBSCRIBE_4.INIT;
        SUBSCRIBE_4.INITO TO SUBSCRIBE_5.INIT;
        SUBSCRIBE_4.IND TO E_SWITCH_2.EI;
        START.COLD TO SUBSCRIBE_9.INIT;
        START.WARM TO SUBSCRIBE_9.INIT;
        CLIENT_0.INITO TO SERVER_4.INIT;
      END_CONNECTIONS
      DATA_CONNECTIONS
        SERVER_2.RD_1 TO AROBOT_MUX.PresetPosition;
        SERVER_3.RD_1 TO ATURNTABLE_MUX.Position;
        ATURNTABLE_MUX.CurrentPosition TO PUBLISH_3.SD_1;
        E_RS_2.Q TO PUBLISH_0.SD_1;
        AROBOT_MUX.CurrentPosition TO PUBLISH_2.SD_1;
        E_RS_3.Q TO PUBLISH_1.SD_1;
        E_RS.Q TO PUBLISH_4.SD_1;
        E_RS_1.Q TO PUBLISH_5.SD_1;
        SUBSCRIBE_9.RD_1 TO E_SWITCH_1.G;
        ATURNTABLE_DEMUX.Position TO CLIENT_2.SD_1;
        SUBSCRIBE_1.RD_1 TO AROBOT_DEMUX.CurrentPosition;
        AROBOT_DEMUX.PresetPosition TO CLIENT_1.SD_1;
        SUBSCRIBE_5.RD_1 TO E_SWITCH_3.G;
        SUBSCRIBE_2.RD_1 TO ATURNTABLE_DEMUX.CurrentPosition;
        SUBSCRIBE_3.RD_1 TO E_SWITCH.G;
        SUBSCRIBE_4.RD_1 TO E_SWITCH_2.G;
      END_CONNECTIONS
      ADAPTER_CONNECTIONS
        AROBOT_MUX.ARobot TO Robot.ARobot;
        ATURNTABLE_MUX.ATurntable TO Turntable.ATurntable;
        AGRIPPER_MUX.AGripper TO Gripper.AGripper;
        ASTORAGE_MUX.AStorage TO Storage.AStorage;
        HandlingControl.AGripper TO AGRIPPER_DEMUX.AGripper;
        DepotControl.ATurntable TO ATURNTABLE_DEMUX.ATurntable;
        HandlingControl.ARobot TO AROBOT_DEMUX.ARobot;
        DepotControl.AStorage TO ASTORAGE_DEMUX.AStorage;
        Station1Control.ADepot TO DepotControl.ADepot;
        Station1Control.AHandling TO HandlingControl.AHandling;
      END_CONNECTIONS
    END_RESOURCE
    RESOURCE skill_decentral : EMB_RES
      FBS
        SERVER_0_1 : SERVER_0_1(QI := 1, ID := opc_ua[CREATE_METHOD;/Objects/4:RobotSkill/4:SetStartParams]);
        SERVER_0_2 : SERVER_0_1(QI := 1, ID := opc_ua[CREATE_METHOD;/Objects/4:TurntableSkill/4:SetStartParams]);
        CLIENT_1_1 : CLIENT_1_0(QI := 1, ID := opc_ua[CALL_METHOD;opc.tcp://localhost:4850#;/Objects/4:RobotSkill/4:SetStartParams]);
        Station1Control : Station1Skill;
        CLIENT_1_0 : CLIENT_1_0(QI := 1, ID := opc_ua[CALL_METHOD;opc.tcp://localhost:4850#;/Objects/4:TurntableSkill/4:SetStartParams]);
      END_FBS
      SUBAPPS
        SServer_2 : SServer(skillName := GripperSkill);
        SServer_3 : SServer(skillName := RobotSkill);
        SServer_1 : SServer(skillName := TurntableSkill);
        SServer : SServer(skillName := StorageSkill);
        SClient_1 : SClient(remoteIPandPort := localhost:4850, IAS_Namespace := STRING#4, skillStateMachineNodeBrowsePath := STRING#4:TurntableSkill/4:StateMachine/);
        SClient : SClient(remoteIPandPort := localhost:4850, IAS_Namespace := STRING#4, skillStateMachineNodeBrowsePath := STRING#4:StorageSkill/4:StateMachine/);
        SClient_3 : SClient(remoteIPandPort := localhost:4850, IAS_Namespace := STRING#4, skillStateMachineNodeBrowsePath := STRING#4:RobotSkill/4:StateMachine/);
        SClient_2 : SClient(remoteIPandPort := localhost:4850, IAS_Namespace := STRING#4, skillStateMachineNodeBrowsePath := STRING#4:GripperSkill/4:StateMachine/);
      END_SUBAPPS
      SUBAPPLICATION RobotSkill
        EVENT_INPUT
          INIT;
          SetStartParam_REQ;
        END_EVENT
        EVENT_OUTPUT
          INITO;
        END_EVENT
        VAR_INPUT
          Robot_SetStartParam_IN : WORD;
        END_VAR
        SOCKETS
          AIAS_Skill : IAS_Skill;
        END_SOCKETS
      END_SUBAPPLICATION
      SUBAPPLICATION TurntableSkill
        EVENT_INPUT
          INIT;
          Table_SetStartParam_REQ;
        END_EVENT
        EVENT_OUTPUT
          INITO;
        END_EVENT
        VAR_INPUT
          Table_SetStartParam_IN : WORD;
        END_VAR
        SOCKETS
          AIAS_Skill : IAS_Skill;
        END_SOCKETS
      END_SUBAPPLICATION
      SUBAPPLICATION StorageSkill
        EVENT_INPUT
          INIT;
        END_EVENT
        EVENT_OUTPUT
          INITO;
        END_EVENT
        SOCKETS
          AIAS_Skill : IAS_Skill;
        END_SOCKETS
      END_SUBAPPLICATION
      SUBAPPLICATION GripperSkill
        EVENT_INPUT
          INIT;
        END_EVENT
        EVENT_OUTPUT
          INITO;
        END_EVENT
        SOCKETS
          AIAS_Skill : IAS_Skill;
        END_SOCKETS
      END_SUBAPPLICATION
      SUBAPPLICATION DepotSkill
        EVENT_INPUT
          INIT;
        END_EVENT
        EVENT_OUTPUT
          INITO;
          TurntablePresetPositionUpd;
        END_EVENT
        VAR_OUTPUT
          TurntablePresetPosition : WORD;
        END_VAR
        SOCKETS
          AIAS_Skill : IAS_Skill;
        END_SOCKETS
        PLUGS
          AIAS_Skill_Storage : IAS_Skill;
          AIAS_Skill_Turntable : IAS_Skill;
        END_PLUGS
      END_SUBAPPLICATION
      SUBAPPLICATION HandlingSkill
        EVENT_INPUT
          INIT;
        END_EVENT
        EVENT_OUTPUT
          INITO;
          RobotPositionUpd;
        END_EVENT
        VAR_OUTPUT
          RobotPresetPosition : WORD;
        END_VAR
        SOCKETS
          AIAS_Skill : IAS_Skill;
        END_SOCKETS
        PLUGS
          AIAS_Skill_Gripper : IAS_Skill;
          AIAS_Skill_Robot : IAS_Skill;
        END_PLUGS
      END_SUBAPPLICATION
      EVENT_CONNECTIONS
        TurntableSkill.INITO TO TurntableSkill.Table_SetStartParam_REQ;
        StorageSkill.INITO TO SServer.INIT;
        GripperSkill.INITO TO SServer_2.INIT;
        START.WARM TO StorageSkill.INIT;
        START.COLD TO StorageSkill.INIT;
        StorageSkill.INITO TO TurntableSkill.INIT;
        TurntableSkill.INITO TO GripperSkill.INIT;
        GripperSkill.INITO TO RobotSkill.INIT;
        SERVER_0_1.IND TO RobotSkill.SetStartParam_REQ;
        SERVER_0_2.IND TO TurntableSkill.Table_SetStartParam_REQ;
        SClient_2.INITO TO CLIENT_1_1.INIT;
        DepotSkill.INITO TO SClient_1.INIT;
        DepotSkill.INITO TO SClient.INIT;
        DepotSkill.INITO TO HandlingSkill.INIT;
        HandlingSkill.INITO TO SClient_3.INIT;
        HandlingSkill.INITO TO SClient_2.INIT;
        HandlingSkill.RobotPositionUpd TO CLIENT_1_1.REQ;
        SClient.INITO TO CLIENT_1_0.INIT;
        DepotSkill.TurntablePresetPositionUpd TO CLIENT_1_0.REQ;
        START.COLD TO DepotSkill.INIT;
        START.WARM TO DepotSkill.INIT;
        SServer.INITO TO SServer_1.INIT;
        RobotSkill.INITO TO SServer_3.INIT;
        SServer_3.INITO TO SERVER_0_1.INIT;
        SServer_1.INITO TO SERVER_0_2.INIT;
        SERVER_0_2.IND TO SERVER_0_2.RSP;
        SERVER_0_1.IND TO SERVER_0_1.RSP;
      END_CONNECTIONS
      DATA_CONNECTIONS
        SERVER_0_1.RD_1 TO RobotSkill.Robot_SetStartParam_IN;
        SERVER_0_2.RD_1 TO TurntableSkill.Table_SetStartParam_IN;
        HandlingSkill.RobotPresetPosition TO CLIENT_1_1.SD_1;
        DepotSkill.TurntablePresetPosition TO CLIENT_1_0.SD_1;
      END_CONNECTIONS
      ADAPTER_CONNECTIONS
        SServer_3.IAS_Skill TO RobotSkill.AIAS_Skill;
        SServer_1.IAS_Skill TO TurntableSkill.AIAS_Skill;
        SServer.IAS_Skill TO StorageSkill.AIAS_Skill;
        SServer_2.IAS_Skill TO GripperSkill.AIAS_Skill;
        DepotSkill.AIAS_Skill_Storage TO SClient.IAS_Skill;
        DepotSkill.AIAS_Skill_Turntable TO SClient_1.IAS_Skill;
        Station1Control.ADepot TO DepotSkill.AIAS_Skill;
        HandlingSkill.AIAS_Skill_Gripper TO SClient_2.IAS_Skill;
        HandlingSkill.AIAS_Skill_Robot TO SClient_3.IAS_Skill;
        Station1Control.AHandling TO HandlingSkill.AIAS_Skill;
      END_CONNECTIONS
    END_RESOURCE
    RESOURCE codegen_decentral : EMB_RES
      FBS
        IAS_SKILL_MUX_GEN : IAS_SKILL_MUX_GEN;
        PUBLISH_2 : PUBLISH_2(QI := 1, ID := opc_ua[WRITE;/Objects/StorageSkill/currentState;/Objects/StorageSkill/lastTransition]);
        SERVER_0 : SERVER_0(QI := 1, ID := opc_ua[CREATE_METHOD;/Objects/StorageSkill/cleanUp,1:s=StorageSkill_cleanUp]);
        SERVER_1 : SERVER_0(QI := 1, ID := opc_ua[CREATE_METHOD;/Objects/StorageSkill/lock,1:s=StorageSkill_lock]);
        SERVER_2 : SERVER_0(QI := 1, ID := opc_ua[CREATE_METHOD;/Objects/StorageSkill/reset,1:s=StorageSkill_reset]);
        SERVER_3 : SERVER_0(QI := 1, ID := opc_ua[CREATE_METHOD;/Objects/StorageSkill/start,1:s=StorageSkill_start]);
        SERVER_4 : SERVER_0(QI := 1, ID := opc_ua[CREATE_METHOD;/Objects/StorageSkill/stop,1:s=StorageSkill_stop]);
        SERVER_5 : SERVER_0(QI := 1, ID := opc_ua[CREATE_METHOD;/Objects/StorageSkill/suspend,1:s=StorageSkill_suspend]);
        SERVER_6 : SERVER_0(QI := 1, ID := opc_ua[CREATE_METHOD;/Objects/StorageSkill/unsuspend,1:s=StorageSkill_unsuspend]);
        SERVER_8 : SERVER_0(QI := 1, ID := opc_ua[CREATE_METHOD;/Objects/TurntableSkill/cleanUp,1:s=TurntableSkill_cleanUp]);
        SERVER_7 : SERVER_0_1(QI := 1, ID := opc_ua[CREATE_METHOD;/Objects/TurnTableSetStartParams/IND,1:s=TurnTableSetStartParams_IND]);
        SERVER_15 : SERVER_0_1(QI := 1, ID := opc_ua[CREATE_METHOD;/Objects/RobotSetStartParams/IND,1:s=RobotSetStartParams_IND]);
        SERVER_14 : SERVER_0(QI := 1, ID := opc_ua[CREATE_METHOD;/Objects/TurntableSkill/unsuspend,1:s=TurntableSkill_unsuspend]);
        SERVER_22 : SERVER_0(QI := 1, ID := opc_ua[CREATE_METHOD;/Objects/RobotSkill/unsuspend,1:s=RobotSkill_unsuspend]);
        SERVER_29 : SERVER_0(QI := 1, ID := opc_ua[CREATE_METHOD;/Objects/GripperSkill/unsuspend,1:s=GripperSkill_unsuspend]);
        SERVER_13 : SERVER_0(QI := 1, ID := opc_ua[CREATE_METHOD;/Objects/TurntableSkill/suspend,1:s=TurntableSkill_suspend]);
        SERVER_21 : SERVER_0(QI := 1, ID := opc_ua[CREATE_METHOD;/Objects/RobotSkill/suspend,1:s=RobotSkill_suspend]);
        SERVER_28 : SERVER_0(QI := 1, ID := opc_ua[CREATE_METHOD;/Objects/GripperSkill/suspend,1:s=GripperSkill_suspend]);
        SERVER_12 : SERVER_0(QI := 1, ID := opc_ua[CREATE_METHOD;/Objects/TurntableSkill/stop,1:s=TurntableSkill_stop]);
        SERVER_20 : SERVER_0(QI := 1, ID := opc_ua[CREATE_METHOD;/Objects/RobotSkill/stop,1:s=RobotSkill_stop]);
        SERVER_27 : SERVER_0(QI := 1, ID := opc_ua[CREATE_METHOD;/Objects/GripperSkill/stop,1:s=GripperSkill_stop]);
        SERVER_11 : SERVER_0(QI := 1, ID := opc_ua[CREATE_METHOD;/Objects/TurntableSkill/start,1:s=TurntableSkill_start]);
        SERVER_19 : SERVER_0(QI := 1, ID := opc_ua[CREATE_METHOD;/Objects/RobotSkill/start,1:s=RobotSkill_start]);
        SERVER_26 : SERVER_0(QI := 1, ID := opc_ua[CREATE_METHOD;/Objects/GripperSkill/start,1:s=GripperSkill_start]);
        SERVER_10 : SERVER_0(QI := 1, ID := opc_ua[CREATE_METHOD;/Objects/TurntableSkill/reset,1:s=TurntableSkill_reset]);
        SERVER_18 : SERVER_0(QI := 1, ID := opc_ua[CREATE_METHOD;/Objects/RobotSkill/reset,1:s=RobotSkill_reset]);
        SERVER_25 : SERVER_0(QI := 1, ID := opc_ua[CREATE_METHOD;/Objects/GripperSkill/reset,1:s=GripperSkill_reset]);
        SERVER_9 : SERVER_0(QI := 1, ID := opc_ua[CREATE_METHOD;/Objects/TurntableSkill/lock,1:s=TurntableSkill_lock]);
        SERVER_17 : SERVER_0(QI := 1, ID := opc_ua[CREATE_METHOD;/Objects/RobotSkill/lock,1:s=RobotSkill_lock]);
        SERVER_24 : SERVER_0(QI := 1, ID := opc_ua[CREATE_METHOD;/Objects/GripperSkill/lock,1:s=GripperSkill_lock]);
        SERVER_16 : SERVER_0(QI := 1, ID := opc_ua[CREATE_METHOD;/Objects/RobotSkill/cleanUp,1:s=RobotSkill_cleanUp]);
        SERVER_23 : SERVER_0(QI := 1, ID := opc_ua[CREATE_METHOD;/Objects/GripperSkill/cleanUp,1:s=GripperSkill_cleanUp]);
        PUBLISH_3 : PUBLISH_2(QI := 1, ID := opc_ua[WRITE;/Objects/TurntableSkill/currentState;/Objects/TurntableSkill/lastTransition]);
        PUBLISH_4 : PUBLISH_2(QI := 1, ID := opc_ua[WRITE;/Objects/RobotSkill/currentState;/Objects/RobotSkill/lastTransition]);
        PUBLISH_5 : PUBLISH_2(QI := 1, ID := opc_ua[WRITE;/Objects/GripperSkill/currentState;/Objects/GripperSkill/lastTransition]);
        SETPARAMS1WORD_MUX_GEN_1 : SETPARAMS1WORD_MUX_GEN;
        SETPARAMS1WORD_MUX_GEN : SETPARAMS1WORD_MUX_GEN;
        IAS_SKILL_MUX_GEN_1 : IAS_SKILL_MUX_GEN;
        IAS_SKILL_MUX_GEN_2 : IAS_SKILL_MUX_GEN;
        IAS_SKILL_MUX_GEN_3 : IAS_SKILL_MUX_GEN;
      END_FBS
      SUBAPPLICATION StorageSkill
        EVENT_INPUT
          INIT;
        END_EVENT
        EVENT_OUTPUT
          INITO;
        END_EVENT
        SOCKETS
          AIAS_Skill : IAS_Skill;
        END_SOCKETS
      END_SUBAPPLICATION
      SUBAPPLICATION GripperSkill
        EVENT_INPUT
          INIT;
        END_EVENT
        EVENT_OUTPUT
          INITO;
        END_EVENT
        SOCKETS
          AIAS_Skill : IAS_Skill;
        END_SOCKETS
      END_SUBAPPLICATION
      SUBAPPLICATION RobotSkill
        EVENT_INPUT
          INIT;
          SetStartParam_REQ;
        END_EVENT
        EVENT_OUTPUT
          INITO;
        END_EVENT
        VAR_INPUT
          Robot_SetStartParam_IN : WORD;
        END_VAR
        SOCKETS
          AIAS_Skill : IAS_Skill;
        END_SOCKETS
      END_SUBAPPLICATION
      SUBAPPLICATION TurntableSkill
        EVENT_INPUT
          INIT;
          Table_SetStartParam_REQ;
        END_EVENT
        EVENT_OUTPUT
          INITO;
        END_EVENT
        VAR_INPUT
          Table_SetStartParam_IN : WORD;
        END_VAR
        SOCKETS
          AIAS_Skill : IAS_Skill;
        END_SOCKETS
      END_SUBAPPLICATION
      SUBAPPLICATION RobotSetStartParams
        EVENT_OUTPUT
          SetParams;
        END_EVENT
        VAR_OUTPUT
          WORD : WORD;
        END_VAR
        SOCKETS
          SetStartParams : SetParams1Word;
        END_SOCKETS
      END_SUBAPPLICATION
      SUBAPPLICATION TurnTableSetStartParams
        EVENT_OUTPUT
          SetParams;
        END_EVENT
        VAR_OUTPUT
          WORD : WORD;
        END_VAR
        SOCKETS
          SetStartParams : SetParams1Word;
        END_SOCKETS
      END_SUBAPPLICATION
      EVENT_CONNECTIONS
        IAS_SKILL_MUX_GEN.RSP TO PUBLISH_2.REQ;
        SERVER_0.IND TO IAS_SKILL_MUX_GEN.cleanUp;
        SERVER_1.IND TO IAS_SKILL_MUX_GEN.lock;
        SERVER_2.IND TO IAS_SKILL_MUX_GEN.reset;
        SERVER_3.IND TO IAS_SKILL_MUX_GEN.start;
        SERVER_4.IND TO IAS_SKILL_MUX_GEN.stop;
        SERVER_5.IND TO IAS_SKILL_MUX_GEN.suspend;
        SERVER_6.IND TO IAS_SKILL_MUX_GEN.unsuspend;
        START.COLD TO SERVER_0.INIT;
        START.WARM TO SERVER_0.INIT;
        SERVER_0.INITO TO SERVER_1.INIT;
        SERVER_1.INITO TO SERVER_2.INIT;
        SERVER_2.INITO TO SERVER_3.INIT;
        SERVER_3.INITO TO SERVER_4.INIT;
        SERVER_4.INITO TO SERVER_5.INIT;
        SERVER_5.INITO TO SERVER_6.INIT;
        SERVER_6.INITO TO PUBLISH_2.INIT;
        SERVER_0.IND TO SERVER_0.RSP;
        SERVER_1.IND TO SERVER_1.RSP;
        SERVER_2.IND TO SERVER_2.RSP;
        SERVER_3.IND TO SERVER_3.RSP;
        SERVER_4.IND TO SERVER_4.RSP;
        SERVER_5.IND TO SERVER_5.RSP;
        SERVER_6.IND TO SERVER_6.RSP;
        START.COLD TO StorageSkill.INIT;
        START.WARM TO StorageSkill.INIT;
        SERVER_8.IND TO SERVER_8.RSP;
        START.WARM TO SERVER_8.INIT;
        START.COLD TO SERVER_8.INIT;
        SERVER_7.IND TO SERVER_7.RSP;
        START.WARM TO SERVER_7.INIT;
        START.COLD TO SERVER_7.INIT;
        SERVER_15.IND TO SERVER_15.RSP;
        START.WARM TO SERVER_15.INIT;
        START.COLD TO SERVER_15.INIT;
        SERVER_14.IND TO SERVER_14.RSP;
        SERVER_22.IND TO SERVER_22.RSP;
        SERVER_29.IND TO SERVER_29.RSP;
        SERVER_13.IND TO SERVER_13.RSP;
        SERVER_13.INITO TO SERVER_14.INIT;
        SERVER_21.IND TO SERVER_21.RSP;
        SERVER_21.INITO TO SERVER_22.INIT;
        SERVER_28.IND TO SERVER_28.RSP;
        SERVER_28.INITO TO SERVER_29.INIT;
        SERVER_12.IND TO SERVER_12.RSP;
        SERVER_12.INITO TO SERVER_13.INIT;
        SERVER_20.IND TO SERVER_20.RSP;
        SERVER_20.INITO TO SERVER_21.INIT;
        SERVER_27.IND TO SERVER_27.RSP;
        SERVER_27.INITO TO SERVER_28.INIT;
        SERVER_11.IND TO SERVER_11.RSP;
        SERVER_11.INITO TO SERVER_12.INIT;
        SERVER_19.IND TO SERVER_19.RSP;
        SERVER_19.INITO TO SERVER_20.INIT;
        SERVER_26.IND TO SERVER_26.RSP;
        SERVER_26.INITO TO SERVER_27.INIT;
        SERVER_10.IND TO SERVER_10.RSP;
        SERVER_10.INITO TO SERVER_11.INIT;
        SERVER_18.IND TO SERVER_18.RSP;
        SERVER_18.INITO TO SERVER_19.INIT;
        SERVER_25.IND TO SERVER_25.RSP;
        SERVER_25.INITO TO SERVER_26.INIT;
        SERVER_9.IND TO SERVER_9.RSP;
        SERVER_9.INITO TO SERVER_10.INIT;
        SERVER_8.INITO TO SERVER_9.INIT;
        SERVER_17.IND TO SERVER_17.RSP;
        SERVER_17.INITO TO SERVER_18.INIT;
        SERVER_24.IND TO SERVER_24.RSP;
        SERVER_24.INITO TO SERVER_25.INIT;
        SERVER_16.IND TO SERVER_16.RSP;
        SERVER_16.INITO TO SERVER_17.INIT;
        START.WARM TO SERVER_16.INIT;
        START.COLD TO SERVER_16.INIT;
        SERVER_23.IND TO SERVER_23.RSP;
        SERVER_23.INITO TO SERVER_24.INIT;
        START.WARM TO SERVER_23.INIT;
        START.COLD TO SERVER_23.INIT;
        SERVER_14.INITO TO PUBLISH_3.INIT;
        SERVER_22.INITO TO PUBLISH_4.INIT;
        SERVER_29.INITO TO PUBLISH_5.INIT;
        SERVER_15.IND TO SETPARAMS1WORD_MUX_GEN_1.IND;
        SERVER_7.IND TO SETPARAMS1WORD_MUX_GEN.IND;
        IAS_SKILL_MUX_GEN_1.RSP TO PUBLISH_3.REQ;
        SERVER_14.IND TO IAS_SKILL_MUX_GEN_1.unsuspend;
        SERVER_13.IND TO IAS_SKILL_MUX_GEN_1.suspend;
        SERVER_12.IND TO IAS_SKILL_MUX_GEN_1.stop;
        SERVER_11.IND TO IAS_SKILL_MUX_GEN_1.start;
        SERVER_10.IND TO IAS_SKILL_MUX_GEN_1.reset;
        SERVER_9.IND TO IAS_SKILL_MUX_GEN_1.lock;
        SERVER_8.IND TO IAS_SKILL_MUX_GEN_1.cleanUp;
        IAS_SKILL_MUX_GEN_2.RSP TO PUBLISH_4.REQ;
        SERVER_22.IND TO IAS_SKILL_MUX_GEN_2.unsuspend;
        SERVER_21.IND TO IAS_SKILL_MUX_GEN_2.suspend;
        SERVER_20.IND TO IAS_SKILL_MUX_GEN_2.stop;
        SERVER_19.IND TO IAS_SKILL_MUX_GEN_2.start;
        SERVER_18.IND TO IAS_SKILL_MUX_GEN_2.reset;
        SERVER_17.IND TO IAS_SKILL_MUX_GEN_2.lock;
        SERVER_16.IND TO IAS_SKILL_MUX_GEN_2.cleanUp;
        IAS_SKILL_MUX_GEN_3.RSP TO PUBLISH_5.REQ;
        SERVER_29.IND TO IAS_SKILL_MUX_GEN_3.unsuspend;
        SERVER_28.IND TO IAS_SKILL_MUX_GEN_3.suspend;
        SERVER_27.IND TO IAS_SKILL_MUX_GEN_3.stop;
        SERVER_26.IND TO IAS_SKILL_MUX_GEN_3.start;
        SERVER_25.IND TO IAS_SKILL_MUX_GEN_3.reset;
        SERVER_24.IND TO IAS_SKILL_MUX_GEN_3.lock;
        SERVER_23.IND TO IAS_SKILL_MUX_GEN_3.cleanUp;
        StorageSkill.INITO TO TurntableSkill.INIT;
        GripperSkill.INITO TO RobotSkill.INIT;
        RobotSetStartParams.SetParams TO RobotSkill.SetStartParam_REQ;
        TurntableSkill.INITO TO GripperSkill.INIT;
        TurnTableSetStartParams.SetParams TO TurntableSkill.Table_SetStartParam_REQ;
      END_CONNECTIONS
      DATA_CONNECTIONS
        IAS_SKILL_MUX_GEN.currentState TO PUBLISH_2.SD_1;
        IAS_SKILL_MUX_GEN.lastTransition TO PUBLISH_2.SD_2;
        SERVER_15.RD_1 TO SETPARAMS1WORD_MUX_GEN_1.DATA;
        SERVER_7.RD_1 TO SETPARAMS1WORD_MUX_GEN.DATA;
        IAS_SKILL_MUX_GEN_1.lastTransition TO PUBLISH_3.SD_2;
        IAS_SKILL_MUX_GEN_1.currentState TO PUBLISH_3.SD_1;
        IAS_SKILL_MUX_GEN_2.lastTransition TO PUBLISH_4.SD_2;
        IAS_SKILL_MUX_GEN_2.currentState TO PUBLISH_4.SD_1;
        IAS_SKILL_MUX_GEN_3.lastTransition TO PUBLISH_5.SD_2;
        IAS_SKILL_MUX_GEN_3.currentState TO PUBLISH_5.SD_1;
        RobotSetStartParams.WORD TO RobotSkill.Robot_SetStartParam_IN;
        TurnTableSetStartParams.WORD TO TurntableSkill.Table_SetStartParam_IN;
      END_CONNECTIONS
      ADAPTER_CONNECTIONS
        IAS_SKILL_MUX_GEN.IAS_Skill TO StorageSkill.AIAS_Skill;
        IAS_SKILL_MUX_GEN_3.IAS_Skill TO GripperSkill.AIAS_Skill;
        IAS_SKILL_MUX_GEN_2.IAS_Skill TO RobotSkill.AIAS_Skill;
        IAS_SKILL_MUX_GEN_1.IAS_Skill TO TurntableSkill.AIAS_Skill;
        SETPARAMS1WORD_MUX_GEN_1.SetParams1Word TO RobotSetStartParams.SetStartParams;
        SETPARAMS1WORD_MUX_GEN.SetParams1Word TO TurnTableSetStartParams.SetStartParams;
      END_CONNECTIONS
    END_RESOURCE
  END_DEVICE
  MAPPINGS
    VDMA_Station1_EmulatorApp.Robot ON Robot.central.Robot;
    VDMA_Station1_EmulatorApp.InnerTable ON InnerTable.central.InnerTable;
    VDMA_Station1_EmulatorApp.Storage ON Storage.central.Storage;
    VDMA_Station1_EmulatorApp.Gripper1 ON Gripper1.central.Gripper1;
    VDMA_Station1_EmulatorApp.Gripper2 ON Gripper2.EMB_RES.Gripper2;
    VDMA_Station1_EmulatorApp.IOs_to_OPCUA ON IOs_to_OPCUA.EMB_RES.IOs_to_OPCUA;
    VDMA_Station1_SkillbasedControl.StorageSkill ON skillControl.central.StorageSkill;
    VDMA_Station1_SkillbasedControl.TurntableSkill ON skillControl.central.TurntableSkill;
    VDMA_Station1_SkillbasedControl.DepotSkill ON skillControl.central.DepotSkill;
    VDMA_Station1_SkillbasedControl.GripperSkill ON skillControl.central.GripperSkill;
    VDMA_Station1_SkillbasedControl.HandlingSkill ON skillControl.central.HandlingSkill;
    VDMA_Station1_SkillbasedControl.Station1Control ON skillControl.central.Station1Control;
    VDMA_Station1_CodeGenTemplate.RobotSetStartParams ON codeGenControl.central.RobotSetStartParams;
    VDMA_Station1_CodeGenTemplate.TurnTableSetStartParams ON codeGenControl.central.TurnTableSetStartParams;
    VDMA_Station1_HierarchicalControl_Distributed.DepotControl ON hierControl.decentral.DepotControl;
    VDMA_Station1_HierarchicalControl_Distributed.Station1Control ON hierControl.decentral.Station1Control;
    VDMA_Station1_HierarchicalControl_Distributed.HandlingControl ON hierControl.decentral.HandlingControl;
    VDMA_Station1_SkillbasedControl_Distributed.HandlingSkill ON skillControl.decentral.HandlingSkill;
    VDMA_Station1_SkillbasedControl_Distributed.DepotSkill ON skillControl.decentral.DepotSkill;
    VDMA_Station1_SkillbasedControl_Distributed.Station1Control ON skillControl.decentral.Station1Control;
    VDMA_Station1_SkillbasedControl_Distributed.GripperSkill ON Gripper1.decentral.GripperSkill;
    VDMA_Station1_HierarchicalControl_Distributed.CLIENT_0 ON hierControl.decentral.CLIENT_0;
    VDMA_Station1_HierarchicalControl_Distributed.CLIENT_5 ON hierControl.decentral.CLIENT_5;
    VDMA_Station1_HierarchicalControl_Distributed.CLIENT_4 ON hierControl.decentral.CLIENT_4;
    VDMA_Station1_HierarchicalControl_Distributed.RobotSubApp ON hierControl.decentral.RobotSubApp;
    VDMA_Station1_HierarchicalControl_Distributed.SUBSCRIBE_1 ON hierControl.decentral.SUBSCRIBE_1;
    VDMA_Station1_HierarchicalControl_Distributed.SUBSCRIBE_2 ON hierControl.decentral.SUBSCRIBE_2;
    VDMA_Station1_HierarchicalControl_Distributed.TurntableSubApp ON hierControl.decentral.TurntableSubApp;
    VDMA_Station1_SkillbasedControl_Distributed.SClient_2 ON skillControl.decentral.SClient_2;
    VDMA_Station1_SkillbasedControl_Distributed.SClient_1 ON skillControl.decentral.SClient_1;
    VDMA_Station1_SkillbasedControl_Distributed.SClient ON skillControl.decentral.SClient;
    VDMA_Station1_SkillbasedControl_Distributed.SClient_3 ON skillControl.decentral.SClient_3;
    VDMA_Station1_CodeGenControl.StorageSkill ON codeGenControl.central.StorageSkill;
    VDMA_Station1_CodeGenControl.TurntableSkill ON codeGenControl.central.TurntableSkill;
    VDMA_Station1_CodeGenControl.GripperSkill ON codeGenControl.central.GripperSkill;
    VDMA_Station1_CodeGenControl.RobotSkill ON codeGenControl.central.RobotSkill;
    VDMA_Station1_CodeGenControl.TurnTableSetStartParams ON codeGenControl.central.TurnTableSetStartParams;
    VDMA_Station1_CodeGenControl.RobotSetStartParams ON codeGenControl.central.RobotSetStartParams;
    VDMA_Station1_CodeGenTemplate.TurntableSkill ON codeGenControl.central.TurntableSkill;
    VDMA_Station1_CodeGenTemplate.GripperSkill ON codeGenControl.central.GripperSkill;
    VDMA_Station1_CodeGenTemplate.RobotSkill ON codeGenControl.central.RobotSkill;
    VDMA_Station1_CodeGenTemplate.StorageSkill ON codeGenControl.central.StorageSkill;
    VDMA_Station1_HierarchicalControl_Distributed.SUBSCRIBE_5 ON hierControl.decentral.SUBSCRIBE_5;
    VDMA_Station1_HierarchicalControl_Distributed.CLIENT_3 ON hierControl.decentral.CLIENT_3;
    VDMA_Station1_HierarchicalControl_Distributed.SUBSCRIBE_9 ON hierControl.decentral.SUBSCRIBE_9;
    VDMA_Station1_HierarchicalControl_Distributed.SUBSCRIBE_4 ON hierControl.decentral.SUBSCRIBE_4;
    VDMA_Station1_HierarchicalControl_Distributed.SUBSCRIBE_3 ON hierControl.decentral.SUBSCRIBE_3;
    VDMA_Station1_HierarchicalControl_Distributed.CLIENT_1 ON hierControl.decentral.CLIENT_1;
    VDMA_Station1_HierarchicalControl_Distributed.CLIENT_2 ON hierControl.decentral.CLIENT_2;
    VDMA_Station1_HierarchicalControl_Distributed.StorageSubApp ON hierControl.decentral.StorageSubApp;
    VDMA_Station1_HierarchicalControl_Distributed.GripperSubApp ON hierControl.decentral.GripperSubApp;
    VDMA_Station1_HierarchicalControl_Distributed.SERVER_1 ON Gripper1.decentral.SERVER_1;
    VDMA_Station1_HierarchicalControl_Distributed.PUBLISH_0 ON Gripper1.decentral.PUBLISH_0;
    VDMA_Station1_HierarchicalControl_Distributed.SERVER_0 ON Gripper1.decentral.SERVER_0;
    VDMA_Station1_HierarchicalControl_Distributed.PUBLISH_1 ON Gripper1.decentral.PUBLISH_1;
    VDMA_Station1_HierarchicalControl_Distributed.GripperInternalLogicSubApp ON Gripper1.decentral.GripperInternalLogicSubApp;
    VDMA_Station1_SkillbasedControl.RobotSkill ON skillControl.central.RobotSkill;
    VDMA_Station1_SkillbasedControl_Distributed.SServer_2 ON Gripper1.decentral.SServer_2;
    VDMA_Station1_HierarchicalControl.HandlingControl ON hierControl.central.HandlingControl;
    VDMA_Station1_HierarchicalControl.DepotControl ON hierControl.central.DepotControl;
    VDMA_Station1_HierarchicalControl.Robot ON hierControl.central.Robot;
    VDMA_Station1_HierarchicalControl.Gripper ON hierControl.central.Gripper;
    VDMA_Station1_HierarchicalControl.Turntable ON hierControl.central.Turntable;
    VDMA_Station1_HierarchicalControl.Storage ON hierControl.central.Storage;
    VDMA_Station1_HierarchicalControl.Station1Control ON hierControl.central.Station1Control;
  END_MAPPINGS
END_SYSTEM
